KUKA KRL program: MyProgram_318().src

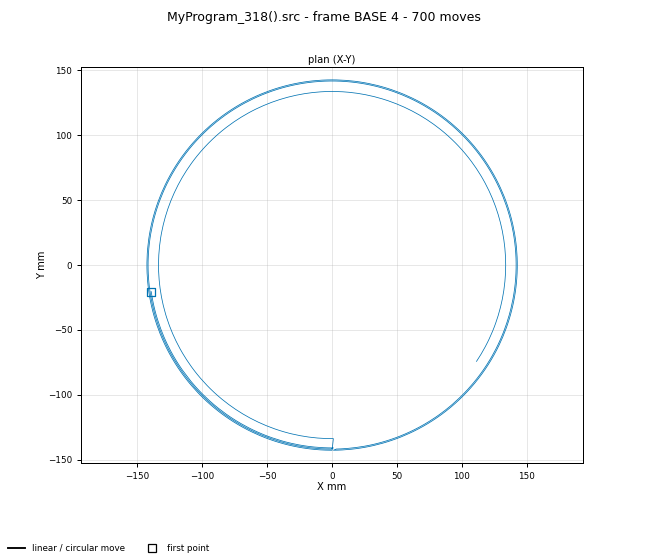
[picture p0: tool path of MyProgram_318().src in frame BASE 4, 700 of 700 moves have a stored position in this frame; points joined in program order, loops and branches not executed]
&ACCESS RVP
&REL 1
&PARAM TEMPLATE = C:\KRC\Roboter\Template\vorgabe
&PARAM EDITMASK = *
DEF MyProgram_318()
; ---- Setting reference (Base) ----
$BASE = BASE_DATA[4]

; --------------------------
; ---- Setting tool (TCP) ----
$TOOL = TOOL_DATA[3]
; --------------------------

$VEL.CP = VEL_APROX_PRINT
Startdeposition()
$VEL.CP = VEL_PRINT
LIN {X -139.4238,Y -20.4254,Z 184,A -166.8954,B 3.5696,C 0.2176,E1 3.4184,E2 259.9212} C_DIS
LIN {X -138.3795,Y -26.5906,Z 184,A -165.0587,B 3.569,C 0.2283,E1 3.4193,E2 258.1802} C_DIS
LIN {X -137.4826,Y -30.8981,Z 184,A -163.1795,B 3.5687,C 0.2327,E1 3.4204,E2 256.2901} C_DIS
LIN {X -136.525,Y -34.8838,Z 184,A -161.5232,B 3.5684,C 0.2373,E1 3.4215,E2 254.636} C_DIS
LIN {X -135.6376,Y -38.1888,Z 184,A -160.0373,B 3.5682,C 0.2406,E1 3.4226,E2 253.1383} C_DIS
LIN {X -134.4577,Y -42.1612,Z 184,A -158.3509,B 3.5678,C 0.2451,E1 3.424,E2 251.4527} C_DIS
LIN {X -131.9427,Y -49.4671,Z 184,A -155.0815,B 3.5673,C 0.2527,E1 3.4271,E2 248.1679} C_DIS
LIN {X -130.7547,Y -52.527,Z 184,A -153.7556,B 3.5671,C 0.2562,E1 3.4284,E2 246.8439} C_DIS
LIN {X -129.4822,Y -55.5908,Z 184,A -152.0943,B 3.5669,C 0.258,E1 3.4303,E2 245.1414} C_DIS
LIN {X -127.3573,Y -60.3009,Z 184,A -150.0342,B 3.5665,C 0.2635,E1 3.4327,E2 243.0877} C_DIS
LIN {X -125.7132,Y -63.6562,Z 184,A -148.6523,B 3.5662,C 0.2681,E1 3.4344,E2 241.7248} C_DIS
LIN {X -124.3831,Y -66.2218,Z 184,A -146.8432,B 3.5662,C 0.2674,E1 3.4368,E2 239.831} C_DIS
LIN {X -122.4083,Y -69.8041,Z 184,A -145.4884,B 3.5658,C 0.2732,E1 3.4386,E2 238.5184} C_DIS
LIN {X -120.1357,Y -73.6466,Z 184,A -143.7295,B 3.5655,C 0.2778,E1 3.4412,E2 236.7677} C_DIS
LIN {X -117.9556,Y -77.0913,Z 184,A -141.8449,B 3.5653,C 0.2803,E1 3.444,E2 234.8531} C_DIS
LIN {X -115.3684,Y -80.9115,Z 184,A -139.9945,B 3.5649,C 0.2847,E1 3.447,E2 233.0067} C_DIS
LIN {X -108.8404,Y -89.5006,Z 184,A -135.5865,B 3.5641,C 0.2942,E1 3.4545,E2 228.5975} C_DIS
LIN {X -105.2184,Y -93.7317,Z 184,A -133.038,B 3.5639,C 0.2971,E1 3.4592,E2 226.0111} C_DIS
LIN {X -102.625,Y -96.5637,Z 184,A -131.4587,B 3.5637,C 0.3001,E1 3.4622,E2 224.4297} C_DIS
LIN {X -99.7736,Y -99.5073,Z 184,A -128.8184,B 3.5639,C 0.2971,E1 3.4678,E2 221.6564} C_DIS
LIN {X -94.4634,Y -104.5617,Z 184,A -126.9429,B 3.5628,C 0.3096,E1 3.4713,E2 219.9326} C_DIS
LIN {X -90.9298,Y -107.6493,Z 184,A -124.7172,B 3.5628,C 0.3109,E1 3.4761,E2 217.664} C_DIS
LIN {X -87.4156,Y -110.5219,Z 184,A -122.849,B 3.5625,C 0.3138,E1 3.4801,E2 215.7928} C_DIS
LIN {X -81.7858,Y -114.7499,Z 184,A -119.9297,B 3.5621,C 0.3179,E1 3.4867,E2 212.866} C_DIS
LIN {X -78.0793,Y -117.3033,Z 184,A -118.0516,B 3.5619,C 0.3203,E1 3.4911,E2 210.9813} C_DIS
LIN {X -74.1308,Y -119.8381,Z 184,A -116.0901,B 3.5617,C 0.3226,E1 3.4957,E2 209.0125} C_DIS
LIN {X -70.4469,Y -122.0396,Z 184,A -114.3288,B 3.5615,C 0.3247,E1 3.5,E2 207.2488} C_DIS
LIN {X -64.5086,Y -125.2793,Z 184,A -111.5655,B 3.5612,C 0.328,E1 3.5068,E2 204.4835} C_DIS
LIN {X -61.1095,Y -126.971,Z 184,A -110.0392,B 3.561,C 0.3298,E1 3.5106,E2 202.9594} C_DIS
LIN {X -57.8227,Y -128.5009,Z 184,A -108.3988,B 3.561,C 0.3301,E1 3.5149,E2 201.296} C_DIS
LIN {X -53.0992,Y -130.5241,Z 184,A -106.388,B 3.5608,C 0.3327,E1 3.52,E2 199.2957} C_DIS
LIN {X -49.9078,Y -131.7776,Z 184,A -105.1272,B 3.5606,C 0.3349,E1 3.5232,E2 198.0529} C_DIS
LIN {X -46.236,Y -133.1094,Z 184,A -102.9524,B 3.5609,C 0.3317,E1 3.5292,E2 195.797} C_DIS
LIN {X -42.002,Y -134.5078,Z 184,A -101.4553,B 3.5605,C 0.3354,E1 3.5331,E2 194.3432} C_DIS
LIN {X -39.0569,Y -135.3911,Z 184,A -100.1869,B 3.5605,C 0.3361,E1 3.5365,E2 193.0719} C_DIS
LIN {X -35.4176,Y -136.3895,Z 184,A -98.6921,B 3.5603,C 0.3373,E1 3.5405,E2 191.5822} C_DIS
LIN {X -31.5759,Y -137.3278,Z 184,A -97.2077,B 3.5602,C 0.3391,E1 3.5445,E2 190.1142} C_DIS
LIN {X -28.2117,Y -138.0581,Z 184,A -95.8313,B 3.5601,C 0.3399,E1 3.5483,E2 188.7406} C_DIS
LIN {X -25.433,Y -138.5982,Z 184,A -94.5046,B 3.5601,C 0.3389,E1 3.552,E2 187.3894} C_DIS
LIN {X -21.5406,Y -139.2549,Z 184,A -92.984,B 3.5601,C 0.34,E1 3.5561,E2 185.8798} C_DIS
LIN {X -17.9488,Y -139.7638,Z 184,A -91.4422,B 3.5601,C 0.3398,E1 3.5604,E2 184.3282} C_DIS
LIN {X -13.5381,Y -140.2594,Z 184,A -89.7378,B 3.56,C 0.3409,E1 3.5651,E2 182.637} C_DIS
LIN {X -10.3708,Y -140.5291,Z 184,A -88.4486,B 3.56,C 0.341,E1 3.5687,E2 181.3477} C_DIS
LIN {X -7.0582,Y -140.7344,Z 184,A -86.9885,B 3.56,C 0.3401,E1 3.5728,E2 179.8718} C_DIS
LIN {X -2.6126,Y -140.8874,Z 184,A -85.2158,B 3.56,C 0.3403,E1 3.5778,E2 178.1032} C_DIS
LIN {X 0.9985,Y -140.9073,Z 184,A -84.3874,B 3.5595,C 0.3456,E1 3.5799,E2 177.3618} C_DIS
Enddeposition()
LIN {X 0.9985,Y -140.9073,Z 184,A -84.3874,B 3.5595,C 0.3456,E1 3.5799,E2 177.3618} C_DIS
Startdeposition()
$VEL.CP = VEL_PRINT
LIN {X -0.7581,Y -141.8102,Z 184,A -85.1116,B 3.5589,C 0.3478,E1 3.5773,E2 178.1199} C_DIS
LIN {X -5.0897,Y -141.7215,Z 184,A -86.9297,B 3.5589,C 0.3485,E1 3.5722,E2 179.9481} C_DIS
LIN {X -9.2783,Y -141.5094,Z 184,A -88.6221,B 3.5589,C 0.3485,E1 3.5675,E2 181.641} C_DIS
LIN {X -13.6823,Y -141.1505,Z 184,A -90.3059,B 3.5589,C 0.3474,E1 3.5628,E2 183.3115} C_DIS
LIN {X -17.2016,Y -140.7655,Z 184,A -91.7391,B 3.5589,C 0.3472,E1 3.5588,E2 184.7456} C_DIS
LIN {X -20.6522,Y -140.3014,Z 184,A -93.2844,B 3.5589,C 0.348,E1 3.5545,E2 186.3106} C_DIS
LIN {X -24.9177,Y -139.6056,Z 184,A -94.9566,B 3.5589,C 0.3468,E1 3.5499,E2 187.9732} C_DIS
LIN {X -28.2573,Y -138.9681,Z 184,A -96.3278,B 3.559,C 0.3463,E1 3.5462,E2 189.3445} C_DIS
LIN {X -32.2456,Y -138.0988,Z 184,A -97.9298,B 3.5591,C 0.3451,E1 3.5418,E2 190.9406} C_DIS
LIN {X -35.6192,Y -137.2678,Z 184,A -99.4409,B 3.5591,C 0.3451,E1 3.5377,E2 192.4668} C_DIS
LIN {X -40.243,Y -135.9825,Z 184,A -101.1414,B 3.5594,C 0.3421,E1 3.5332,E2 194.1351} C_DIS
LIN {X -46.7478,Y -133.8854,Z 184,A -104.5205,B 3.5592,C 0.3448,E1 3.524,E2 197.5994} C_DIS
LIN {X -50.6351,Y -132.4661,Z 184,A -105.7791,B 3.5596,C 0.3403,E1 3.5209,E2 198.802} C_DIS
LIN {X -53.5532,Y -131.3123,Z 184,A -107.0843,B 3.5596,C 0.3394,E1 3.5175,E2 200.1125} C_DIS
LIN {X -56.8322,Y -129.9269,Z 184,A -108.5455,B 3.5598,C 0.3381,E1 3.5137,E2 201.5771} C_DIS
LIN {X -59.8555,Y -128.5612,Z 184,A -109.9347,B 3.5599,C 0.3371,E1 3.5102,E2 202.9731} C_DIS
LIN {X -63.1305,Y -126.9853,Z 184,A -111.4004,B 3.5601,C 0.3354,E1 3.5065,E2 204.4386} C_DIS
LIN {X -66.721,Y -125.1383,Z 184,A -113.2184,B 3.5601,C 0.3349,E1 3.5019,E2 206.2823} C_DIS
LIN {X -70.8009,Y -122.8756,Z 184,A -115.1047,B 3.5603,C 0.3325,E1 3.4973,E2 208.1689} C_DIS
LIN {X -74.881,Y -120.4323,Z 184,A -117.0229,B 3.5606,C 0.3299,E1 3.4927,E2 210.0867} C_DIS
LIN {X -78.6833,Y -117.9832,Z 184,A -118.8829,B 3.5608,C 0.3275,E1 3.4884,E2 211.9511} C_DIS
LIN {X -82.4224,Y -115.4021,Z 184,A -120.7734,B 3.561,C 0.3251,E1 3.484,E2 213.8491} C_DIS
LIN {X -86.4102,Y -112.4477,Z 184,A -122.695,B 3.5614,C 0.3213,E1 3.4798,E2 215.7593} C_DIS
LIN {X -89.4085,Y -110.079,Z 184,A -124.4431,B 3.5614,C 0.3201,E1 3.4759,E2 217.5349} C_DIS
LIN {X -93.1808,Y -106.9039,Z 184,A -126.2519,B 3.5619,C 0.3155,E1 3.4721,E2 219.3188} C_DIS
LIN {X -95.7019,Y -104.6536,Z 184,A -127.8582,B 3.5619,C 0.3145,E1 3.4687,E2 220.9575} C_DIS
LIN {X -100.0347,Y -100.5194,Z 184,A -129.9787,B 3.5625,C 0.3082,E1 3.4645,E2 223.0372} C_DIS
LIN {X -103.5928,Y -96.8488,Z 184,A -132.3732,B 3.5627,C 0.3062,E1 3.4598,E2 225.4759} C_DIS
LIN {X -106.2873,Y -93.8834,Z 184,A -134.2151,B 3.5629,C 0.3042,E1 3.4563,E2 227.3476} C_DIS
LIN {X -109.471,Y -90.1518,Z 184,A -136.1691,B 3.5632,C 0.2999,E1 3.4528,E2 229.2974} C_DIS
LIN {X -112.3501,Y -86.5374,Z 184,A -138.4908,B 3.5633,C 0.2986,E1 3.4487,E2 231.6796} C_DIS
LIN {X -114.9652,Y -83.0311,Z 184,A -139.6861,B 3.5639,C 0.2913,E1 3.4469,E2 232.7977} C_DIS
LIN {X -116.9685,Y -80.184,Z 184,A -141.3736,B 3.5641,C 0.2898,E1 3.4441,E2 234.5225} C_DIS
LIN {X -119.5805,Y -76.2344,Z 184,A -143.3398,B 3.5644,C 0.2857,E1 3.4411,E2 236.4953} C_DIS
LIN {X -121.8868,Y -72.4895,Z 184,A -145.1675,B 3.5647,C 0.2818,E1 3.4385,E2 238.3292} C_DIS
LIN {X -124.1077,Y -68.6177,Z 184,A -147.1404,B 3.565,C 0.2784,E1 3.4357,E2 240.324} C_DIS
LIN {X -125.7385,Y -65.5782,Z 184,A -148.4282,B 3.5653,C 0.2744,E1 3.4341,E2 241.5971} C_DIS
LIN {X -127.3592,Y -62.3725,Z 184,A -149.9746,B 3.5655,C 0.2713,E1 3.4321,E2 243.1556} C_DIS
LIN {X -129.5232,Y -57.7435,Z 184,A -152.0254,B 3.5659,C 0.266,E1 3.4298,E2 245.2037} C_DIS
LIN {X -131.0036,Y -54.3023,Z 184,A -153.6597,B 3.5662,C 0.2628,E1 3.428,E2 246.8533} C_DIS
LIN {X -132.4612,Y -50.6478,Z 184,A -155.2899,B 3.5664,C 0.2588,E1 3.4263,E2 248.4883} C_DIS
LIN {X -133.7803,Y -47.0508,Z 184,A -157.1342,B 3.5666,C 0.2563,E1 3.4245,E2 250.3712} C_DIS
LIN {X -135.5727,Y -41.6009,Z 184,A -159.3512,B 3.5671,C 0.2496,E1 3.4227,E2 252.5735} C_DIS
LIN {X -136.6568,Y -37.8891,Z 184,A -160.9424,B 3.5674,C 0.2456,E1 3.4214,E2 254.1677} C_DIS
LIN {X -137.5543,Y -34.4901,Z 184,A -162.3548,B 3.5677,C 0.2417,E1 3.4204,E2 255.5783} C_DIS
LIN {X -138.2758,Y -31.4708,Z 184,A -163.6845,B 3.5679,C 0.2386,E1 3.4196,E2 256.9172} C_DIS
LIN {X -138.9436,Y -28.3779,Z 184,A -165.4551,B 3.5679,C 0.2376,E1 3.4186,E2 258.752} C_DIS
LIN {X -139.7115,Y -24.3262,Z 184,A -166.9229,B 3.5683,C 0.232,E1 3.4179,E2 260.1928} C_DIS
LIN {X -140.4101,Y -19.891,Z 184,A -168.6787,B 3.5686,C 0.2267,E1 3.4171,E2 261.9398} C_DIS
LIN {X -140.9297,Y -15.8077,Z 184,A -170.7984,B 3.5688,C 0.2243,E1 3.4164,E2 264.1183} C_DIS
LIN {X -141.3049,Y -11.9832,Z 184,A -172.0737,B 3.5691,C 0.2186,E1 3.4161,E2 265.3564} C_DIS
LIN {X -141.646,Y -6.8675,Z 184,A -174.0827,B 3.5695,C 0.2124,E1 3.4158,E2 267.3558} C_DIS
LIN {X -141.7651,Y -3.6623,Z 184,A -175.5929,B 3.5697,C 0.2098,E1 3.4157,E2 268.8933} C_DIS
LIN {X -141.8131,Y 0.1767,Z 184,A -177.0204,B 3.57,C 0.2048,E1 3.4157,E2 270.3036} C_DIS
LIN {X -141.7682,Y 3.5529,Z 184,A -178.6647,B 3.57,C 0.2024,E1 3.4157,E2 271.9835} C_DIS
LIN {X -141.5831,Y 8.0813,Z 184,A 179.6286,B 3.5704,C 0.1966,E1 3.4159,E2 273.6727} C_DIS
LIN {X -141.239,Y 12.7605,Z 184,A 177.393,B 3.5706,C 0.193,E1 3.4165,E2 275.9514} C_DIS
LIN {X -140.7795,Y 17.0836,Z 184,A 175.767,B 3.5709,C 0.1874,E1 3.417,E2 277.559} C_DIS
LIN {X -140.3004,Y 20.659,Z 184,A 174.0083,B 3.571,C 0.1848,E1 3.4177,E2 279.3558} C_DIS
LIN {X -139.7122,Y 24.3224,Z 184,A 172.7327,B 3.5713,C 0.1795,E1 3.4182,E2 280.6013} C_DIS
LIN {X -138.1438,Y 32.0486,Z 184,A 169.8477,B 3.5718,C 0.1692,E1 3.4198,E2 283.4451} C_DIS
LIN {X -137.0717,Y 36.3588,Z 184,A 167.4127,B 3.5718,C 0.1675,E1 3.4215,E2 285.9619} C_DIS
LIN {X -136.0472,Y 40.0221,Z 184,A 165.8748,B 3.5721,C 0.1634,E1 3.4227,E2 287.4988} C_DIS
LIN {X -135.0231,Y 43.3519,Z 184,A 164.3959,B 3.5722,C 0.1599,E1 3.4239,E2 288.9859} C_DIS
LIN {X -133.8089,Y 46.9684,Z 184,A 162.8175,B 3.5724,C 0.156,E1 3.4254,E2 290.5678} C_DIS
LIN {X -132.5738,Y 50.3504,Z 184,A 161.3061,B 3.5726,C 0.1525,E1 3.4269,E2 292.0854} C_DIS
LIN {X -131.2818,Y 53.6289,Z 184,A 159.8333,B 3.5727,C 0.149,E1 3.4284,E2 293.5634} C_DIS
LIN {X -130.0287,Y 56.5967,Z 184,A 158.4531,B 3.5728,C 0.146,E1 3.4299,E2 294.9527} C_DIS
LIN {X -128.4997,Y 59.9885,Z 184,A 156.9056,B 3.573,C 0.1424,E1 3.4317,E2 296.5047} C_DIS
LIN {X -127.0221,Y 63.0558,Z 184,A 155.4507,B 3.5731,C 0.1393,E1 3.4335,E2 297.9686} C_DIS
LIN {X -124.9043,Y 67.1567,Z 184,A 153.6487,B 3.5733,C 0.1344,E1 3.4358,E2 299.7612} C_DIS
LIN {X -123.1361,Y 70.3464,Z 184,A 151.9399,B 3.5733,C 0.132,E1 3.4382,E2 301.4989} C_DIS
LIN {X -120.8558,Y 74.1956,Z 184,A 150.0674,B 3.5735,C 0.128,E1 3.4409,E2 303.3783} C_DIS
LIN {X -118.5023,Y 77.8994,Z 184,A 148.0646,B 3.5736,C 0.1251,E1 3.444,E2 305.4089} C_DIS
LIN {X -115.6188,Y 82.1194,Z 184,A 146.0636,B 3.5738,C 0.12,E1 3.4472,E2 307.4001} C_DIS
LIN {X -112.9327,Y 85.7759,Z 184,A 144.1658,B 3.5739,C 0.1163,E1 3.4504,E2 309.3047} C_DIS
LIN {X -110.048,Y 89.4466,Z 184,A 142.3457,B 3.5741,C 0.1118,E1 3.4535,E2 311.1149} C_DIS
LIN {X -107.6501,Y 92.3182,Z 184,A 140.6682,B 3.5741,C 0.1095,E1 3.4566,E2 312.8123} C_DIS
LIN {X -104.3096,Y 96.0761,Z 184,A 138.8317,B 3.5743,C 0.1043,E1 3.46,E2 314.6225} C_DIS
LIN {X -102.1234,Y 98.3973,Z 184,A 137.2326,B 3.5743,C 0.1034,E1 3.4631,E2 316.26} C_DIS
LIN {X -98.7745,Y 101.7581,Z 184,A 135.333,B 3.5744,C 0.0996,E1 3.4669,E2 318.1559} C_DIS
LIN {X -95.6925,Y 104.6622,Z 184,A 133.5206,B 3.5745,C 0.097,E1 3.4706,E2 319.9798} C_DIS
LIN {X -93.0387,Y 107.0279,Z 184,A 132.0732,B 3.5745,C 0.0945,E1 3.4737,E2 321.4276} C_DIS
LIN {X -89.5567,Y 109.9579,Z 184,A 130.1655,B 3.5746,C 0.0917,E1 3.4778,E2 323.3426} C_DIS
LIN {X -85.9082,Y 112.8316,Z 184,A 128.3025,B 3.5747,C 0.0885,E1 3.4819,E2 325.2025} C_DIS
LIN {X -82.2961,Y 115.4924,Z 184,A 126.3982,B 3.5747,C 0.0861,E1 3.4862,E2 327.1171} C_DIS
LIN {X -78.4994,Y 118.106,Z 184,A 124.612,B 3.5749,C 0.0828,E1 3.4903,E2 328.8923} C_DIS
LIN {X -75.2879,Y 120.1791,Z 184,A 122.8858,B 3.5749,C 0.0817,E1 3.4945,E2 330.6403} C_DIS
LIN {X -70.6565,Y 122.9592,Z 184,A 120.7996,B 3.5749,C 0.0781,E1 3.4994,E2 332.7129} C_DIS
LIN {X -67.3455,Y 124.8028,Z 184,A 119.1375,B 3.5749,C 0.077,E1 3.5036,E2 334.3904} C_DIS
LIN {X -63.8671,Y 126.6167,Z 184,A 117.3142,B 3.5749,C 0.0766,E1 3.5082,E2 336.2424} C_DIS
LIN {X -60.8905,Y 128.074,Z 184,A 116.2429,B 3.5751,C 0.0734,E1 3.5108,E2 337.2792} C_DIS
LIN {X -57.6601,Y 129.5605,Z 184,A 114.759,B 3.5751,C 0.0721,E1 3.5146,E2 338.7681} C_DIS
LIN {X -54.3227,Y 130.9951,Z 184,A 113.2583,B 3.5751,C 0.0708,E1 3.5184,E2 340.272} C_DIS
LIN {X -50.7357,Y 132.427,Z 184,A 111.1717,B 3.5751,C 0.073,E1 3.5241,E2 342.4234} C_DIS
LIN {X -46.357,Y 134.0209,Z 184,A 109.7766,B 3.5751,C 0.068,E1 3.5276,E2 343.7564} C_DIS
LIN {X -42.4916,Y 135.2979,Z 184,A 108.1605,B 3.5751,C 0.0665,E1 3.5319,E2 345.368} C_DIS
LIN {X -39.0206,Y 136.3403,Z 184,A 106.3392,B 3.5751,C 0.068,E1 3.5369,E2 347.2332} C_DIS
LIN {X -35.6094,Y 137.2702,Z 184,A 105.2757,B 3.5752,C 0.0645,E1 3.5396,E2 348.2501} C_DIS
LIN {X -31.0466,Y 138.3727,Z 184,A 103.3247,B 3.5752,C 0.0639,E1 3.5449,E2 350.2069} C_DIS
LIN {X -27.2162,Y 139.1771,Z 184,A 101.1819,B 3.5752,C 0.0673,E1 3.551,E2 352.419} C_DIS
LIN {X -22.493,Y 140.0187,Z 184,A 99.5827,B 3.5752,C 0.064,E1 3.5553,E2 353.9748} C_DIS
LIN {X -17.751,Y 140.6983,Z 184,A 97.7622,B 3.5752,C 0.0626,E1 3.5603,E2 355.78} C_DIS
LIN {X -13.7012,Y 141.1487,Z 184,A 96.1311,B 3.5752,C 0.0622,E1 3.5648,E2 357.4083} C_DIS
LIN {X -9.471,Y 141.4975,Z 184,A 94.2713,B 3.5752,C 0.0631,E1 3.57,E2 359.2855} C_DIS
LIN {X -5.7272,Y 141.6966,Z 184,A 92.8784,B 3.5752,C 0.0621,E1 3.5739,E2 360.6624} C_DIS
LIN {X -1.3489,Y 141.8069,Z 184,A 91.1035,B 3.5752,C 0.0623,E1 3.5789,E2 362.4373} C_DIS
LIN {X 2.3537,Y 141.7926,Z 184,A 89.6494,B 3.5752,C 0.0621,E1 3.5829,E2 363.8855} C_DIS
LIN {X 6.5238,Y 141.6632,Z 184,A 87.8816,B 3.5752,C 0.0631,E1 3.5879,E2 365.6629} C_DIS
LIN {X 10.4865,Y 141.4239,Z 184,A 86.3928,B 3.5752,C 0.0626,E1 3.592,E2 367.1366} C_DIS
LIN {X 14.6588,Y 141.0533,Z 184,A 84.6233,B 3.5752,C 0.0639,E1 3.5969,E2 368.9152} C_DIS
LIN {X 18.435,Y 140.6086,Z 184,A 83.1856,B 3.5752,C 0.0638,E1 3.6009,E2 370.34} C_DIS
LIN {X 22.252,Y 140.0564,Z 184,A 81.6384,B 3.5752,C 0.0645,E1 3.6051,E2 371.8853} C_DIS
LIN {X 25.9323,Y 139.4225,Z 184,A 80.0467,B 3.5752,C 0.0661,E1 3.6096,E2 373.487} C_DIS
LIN {X 30.0417,Y 138.5933,Z 184,A 78.4442,B 3.5752,C 0.0664,E1 3.6139,E2 375.0775} C_DIS
LIN {X 34.067,Y 137.6616,Z 184,A 76.5458,B 3.5752,C 0.0697,E1 3.6191,E2 377.0043} C_DIS
LIN {X 37.236,Y 136.8378,Z 184,A 75.5319,B 3.5752,C 0.0681,E1 3.6218,E2 377.9791} C_DIS
LIN {X 43.0876,Y 135.1075,Z 184,A 72.6176,B 3.575,C 0.0743,E1 3.6297,E2 380.9492} C_DIS
LIN {X 47.3667,Y 133.6696,Z 184,A 71.319,B 3.5751,C 0.0714,E1 3.633,E2 382.1814} C_DIS
LIN {X 50.32,Y 132.5852,Z 184,A 70.0377,B 3.5751,C 0.0729,E1 3.6363,E2 383.4638} C_DIS
LIN {X 53.5602,Y 131.3095,Z 184,A 68.6098,B 3.5751,C 0.0747,E1 3.64,E2 384.8941} C_DIS
LIN {X 56.7669,Y 129.9551,Z 184,A 67.2856,B 3.5751,C 0.0756,E1 3.6434,E2 386.2078} C_DIS
LIN {X 59.8342,Y 128.5711,Z 184,A 65.8968,B 3.575,C 0.0776,E1 3.6469,E2 387.6001} C_DIS
LIN {X 63.2915,Y 126.9058,Z 184,A 64.4015,B 3.575,C 0.0791,E1 3.6507,E2 389.0883} C_DIS
LIN {X 66.8063,Y 125.0925,Z 184,A 62.7191,B 3.5749,C 0.0821,E1 3.6549,E2 390.7813} C_DIS
LIN {X 70.8243,Y 122.8621,Z 184,A 60.9061,B 3.5749,C 0.0844,E1 3.6593,E2 392.5886} C_DIS
LIN {X 74.6858,Y 120.5538,Z 184,A 59.1267,B 3.5748,C 0.0868,E1 3.6635,E2 394.3632} C_DIS
LIN {X 78.4315,Y 118.1513,Z 184,A 57.4145,B 3.5748,C 0.0889,E1 3.6675,E2 396.0646} C_DIS
LIN {X 81.9336,Y 115.7499,Z 184,A 55.6871,B 3.5746,C 0.0919,E1 3.6714,E2 397.7934} C_DIS
LIN {X 84.8953,Y 113.5955,Z 184,A 54.2829,B 3.5746,C 0.0937,E1 3.6746,E2 399.1881} C_DIS
LIN {X 88.4894,Y 110.8187,Z 184,A 52.4477,B 3.5746,C 0.097,E1 3.6786,E2 401.0235} C_DIS
LIN {X 92.1059,Y 107.8318,Z 184,A 50.6397,B 3.5744,C 0.0997,E1 3.6824,E2 402.8206} C_DIS
LIN {X 95.439,Y 104.8929,Z 184,A 48.8214,B 3.5744,C 0.1034,E1 3.6862,E2 404.642} C_DIS
LIN {X 98.8945,Y 101.642,Z 184,A 47.024,B 3.5742,C 0.106,E1 3.6898,E2 406.4245} C_DIS
LIN {X 102.1017,Y 98.4196,Z 184,A 45.2316,B 3.5742,C 0.1093,E1 3.6933,E2 408.2115} C_DIS
LIN {X 105.1426,Y 95.1639,Z 184,A 43.493,B 3.574,C 0.1125,E1 3.6966,E2 409.9426} C_DIS
LIN {X 108.1815,Y 91.6946,Z 184,A 41.6738,B 3.574,C 0.1161,E1 3.6999,E2 411.7566} C_DIS
LIN {X 111.1562,Y 88.0653,Z 184,A 39.7825,B 3.5738,C 0.1203,E1 3.7032,E2 413.6478} C_DIS
LIN {X 113.9616,Y 84.4037,Z 184,A 38.0457,B 3.5737,C 0.1232,E1 3.7061,E2 415.3687} C_DIS
LIN {X 116.6457,Y 80.6539,Z 184,A 36.2393,B 3.5736,C 0.127,E1 3.709,E2 417.1684} C_DIS
LIN {X 119.0779,Y 77.017,Z 184,A 34.5492,B 3.5734,C 0.1303,E1 3.7116,E2 418.8491} C_DIS
LIN {X 121.3791,Y 73.3363,Z 184,A 32.8628,B 3.5734,C 0.1339,E1 3.7141,E2 420.5273} C_DIS
LIN {X 123.5885,Y 69.5484,Z 184,A 31.1169,B 3.5732,C 0.138,E1 3.7165,E2 422.2705} C_DIS
LIN {X 125.7362,Y 65.5825,Z 184,A 29.454,B 3.573,C 0.1408,E1 3.7186,E2 423.9134} C_DIS
LIN {X 127.3091,Y 62.4741,Z 184,A 28.0813,B 3.573,C 0.144,E1 3.7203,E2 425.2823} C_DIS
LIN {X 128.8911,Y 59.1422,Z 184,A 26.6443,B 3.5728,C 0.1472,E1 3.722,E2 426.713} C_DIS
LIN {X 130.3679,Y 55.8122,Z 184,A 25.2416,B 3.5727,C 0.1503,E1 3.7236,E2 428.1074} C_DIS
LIN {X 131.7718,Y 52.4133,Z 184,A 23.8217,B 3.5725,C 0.1535,E1 3.7251,E2 429.5194} C_DIS
LIN {X 133.0746,Y 49.0132,Z 184,A 22.3927,B 3.5724,C 0.1569,E1 3.7265,E2 430.9436} C_DIS
LIN {X 134.2106,Y 45.8097,Z 184,A 21.0727,B 3.5722,C 0.16,E1 3.7277,E2 432.2573} C_DIS
LIN {X 135.2039,Y 42.7857,Z 184,A 19.7954,B 3.5721,C 0.1634,E1 3.7288,E2 433.5341} C_DIS
LIN {X 136.5763,Y 38.1771,Z 184,A 17.9257,B 3.5719,C 0.1678,E1 3.7302,E2 435.3953} C_DIS
LIN {X 137.5376,Y 34.5558,Z 184,A 16.4903,B 3.5717,C 0.1711,E1 3.7312,E2 436.8213} C_DIS
LIN {X 138.4117,Y 30.8758,Z 184,A 14.9257,B 3.5715,C 0.1757,E1 3.7322,E2 438.3916} C_DIS
LIN {X 139.5625,Y 25.1588,Z 184,A 12.7711,B 3.5713,C 0.18,E1 3.7333,E2 440.521} C_DIS
LIN {X 140.1862,Y 21.4138,Z 184,A 11.2596,B 3.5711,C 0.184,E1 3.734,E2 442.0304} C_DIS
LIN {X 140.7594,Y 17.2527,Z 184,A 9.5729,B 3.5708,C 0.1886,E1 3.7346,E2 443.7168} C_DIS
LIN {X 141.1688,Y 13.4917,Z 184,A 8.1633,B 3.5707,C 0.1916,E1 3.735,E2 445.1117} C_DIS
LIN {X 141.495,Y 9.5104,Z 184,A 6.4959,B 3.5704,C 0.1967,E1 3.7354,E2 446.7873} C_DIS
LIN {X 141.7161,Y 5.2276,Z 184,A 4.9188,B 3.5702,C 0.1999,E1 3.7356,E2 448.345} C_DIS
LIN {X 141.8087,Y 1.0186,Z 184,A 3.3066,B 3.57,C 0.2037,E1 3.7356,E2 449.9465} C_DIS
LIN {X 141.7901,Y -2.5054,Z 184,A 1.951,B 3.5698,C 0.2069,E1 3.7356,E2 451.2942} C_DIS
LIN {X 141.6567,Y -6.6532,Z 184,A 0.2503,B 3.5695,C 0.2119,E1 3.7354,E2 452.9992} C_DIS
LIN {X 141.4207,Y -10.5304,Z 184,A -1.1819,B 3.5694,C 0.2148,E1 3.7351,E2 454.4143} C_DIS
LIN {X 141.0452,Y -14.7346,Z 184,A -2.9015,B 3.5691,C 0.2198,E1 3.7347,E2 456.137} C_DIS
LIN {X 140.6026,Y -18.4812,Z 184,A -4.2754,B 3.5689,C 0.2223,E1 3.7342,E2 457.492} C_DIS
LIN {X 140.0659,Y -22.1904,Z 184,A -5.7496,B 3.5687,C 0.2261,E1 3.7336,E2 458.9621} C_DIS
LIN {X 139.3696,Y -26.2089,Z 184,A -7.3723,B 3.5684,C 0.2304,E1 3.7328,E2 460.5826} C_DIS
LIN {X 138.4697,Y -30.6145,Z 184,A -9.0357,B 3.5682,C 0.2337,E1 3.7318,E2 462.227} C_DIS
LIN {X 137.8173,Y -33.422,Z 184,A -10.1817,B 3.568,C 0.2367,E1 3.7311,E2 463.3714} C_DIS
LIN {X 136.4961,Y -38.464,Z 184,A -12.2228,B 3.5676,C 0.2418,E1 3.7296,E2 465.4054} C_DIS
LIN {X 134.6511,Y -44.4944,Z 184,A -14.8786,B 3.5671,C 0.2499,E1 3.7274,E2 468.0777} C_DIS
LIN {X 132.5838,Y -50.3236,Z 184,A -17.0608,B 3.5669,C 0.253,E1 3.7253,E2 470.2195} C_DIS
LIN {X 131.3722,Y -53.4046,Z 184,A -18.3931,B 3.5666,C 0.2565,E1 3.724,E2 471.5522} C_DIS
LIN {X 129.6366,Y -57.49,Z 184,A -20.292,B 3.5662,C 0.2624,E1 3.7218,E2 473.4666} C_DIS
LIN {X 127.7631,Y -61.5412,Z 184,A -21.8421,B 3.5661,C 0.2642,E1 3.72,E2 474.9842} C_DIS
LIN {X 126.2478,Y -64.5917,Z 184,A -23.1637,B 3.5658,C 0.2671,E1 3.7184,E2 476.2996} C_DIS
LIN {X 123.295,Y -70.0678,Z 184,A -25.5094,B 3.5655,C 0.2716,E1 3.7153,E2 478.6248} C_DIS
LIN {X 121.5366,Y -73.076,Z 184,A -27.0493,B 3.5651,C 0.2765,E1 3.713,E2 480.1837} C_DIS
LIN {X 119.1386,Y -76.9235,Z 184,A -28.8197,B 3.5648,C 0.2803,E1 3.7104,E2 481.9473} C_DIS
LIN {X 116.6918,Y -80.5871,Z 184,A -30.5138,B 3.5646,C 0.2836,E1 3.7078,E2 483.6313} C_DIS
LIN {X 114.2062,Y -84.0718,Z 184,A -32.2569,B 3.5642,C 0.2878,E1 3.7049,E2 485.3777} C_DIS
LIN {X 111.9161,Y -87.0974,Z 184,A -33.6922,B 3.564,C 0.2903,E1 3.7025,E2 486.801} C_DIS
LIN {X 109.05,Y -90.6602,Z 184,A -36.2224,B 3.5631,C 0.3018,E1 3.6978,E2 489.4247} C_DIS
LIN {X 104.7171,Y -95.6327,Z 184,A -37.9514,B 3.5634,C 0.2975,E1 3.6948,E2 491.0298} C_DIS
LIN {X 102.145,Y -98.3749,Z 184,A -39.5733,B 3.5631,C 0.3018,E1 3.6916,E2 492.6669} C_DIS
LIN {X 98.3692,Y -102.1506,Z 184,A -41.8051,B 3.5626,C 0.3071,E1 3.6872,E2 494.9105} C_DIS
LIN {X 93.0128,Y -107.0505,Z 184,A -44.2498,B 3.5626,C 0.3077,E1 3.6822,E2 497.2911} C_DIS
LIN {X 90.6834,Y -109.0308,Z 184,A -45.7128,B 3.5622,C 0.3125,E1 3.679,E2 498.7862} C_DIS
LIN {X 87.0751,Y -111.9334,Z 184,A -47.5792,B 3.5619,C 0.3159,E1 3.6749,E2 500.6534} C_DIS
LIN {X 82.6246,Y -115.2575,Z 184,A -49.6349,B 3.5617,C 0.3179,E1 3.6704,E2 502.6851} C_DIS
LIN {X 79.8515,Y -117.1965,Z 184,A -51.6427,B 3.5609,C 0.3268,E1 3.6655,E2 504.7812} C_DIS
LIN {X 75.0709,Y -120.3141,Z 184,A -53.6443,B 3.5609,C 0.3274,E1 3.6609,E2 506.7433} C_DIS
LIN {X 71.3861,Y -122.5368,Z 184,A -55.0283,B 3.5609,C 0.3265,E1 3.6577,E2 508.0803} C_DIS
LIN {X 67.317,Y -124.8181,Z 184,A -56.8303,B 3.5607,C 0.3284,E1 3.6533,E2 509.8725} C_DIS
LIN {X 63.4428,Y -126.8312,Z 184,A -58.4524,B 3.5607,C 0.3295,E1 3.6493,E2 511.4764} C_DIS
LIN {X 60.3215,Y -128.3455,Z 184,A -60.3103,B 3.56,C 0.3359,E1 3.6444,E2 513.3977} C_DIS
LIN {X 56.5063,Y -130.0678,Z 184,A -61.3013,B 3.5605,C 0.3311,E1 3.6421,E2 514.294} C_DIS
LIN {X 52.6238,Y -131.687,Z 184,A -63.2158,B 3.5601,C 0.3353,E1 3.6371,E2 516.2393} C_DIS
LIN {X 49.3829,Y -132.9362,Z 184,A -64.603,B 3.5599,C 0.3367,E1 3.6335,E2 517.6252} C_DIS
LIN {X 44.5518,Y -134.632,Z 184,A -66.6349,B 3.5598,C 0.3386,E1 3.6281,E2 519.6534} C_DIS
LIN {X 40.4313,Y -135.9274,Z 184,A -68.515,B 3.5595,C 0.3415,E1 3.623,E2 521.5533} C_DIS
LIN {X 35.9286,Y -137.1865,Z 184,A -70.1982,B 3.5595,C 0.3412,E1 3.6186,E2 523.2094} C_DIS
LIN {X 32.2158,Y -138.1056,Z 184,A -71.7743,B 3.5594,C 0.3428,E1 3.6143,E2 524.7907} C_DIS
LIN {X 28.5507,Y -138.9084,Z 184,A -73.2669,B 3.5593,C 0.3437,E1 3.6102,E2 526.281} C_DIS
LIN {X 24.7544,Y -139.6348,Z 184,A -74.7465,B 3.5593,C 0.3439,E1 3.6062,E2 527.7502} C_DIS
LIN {X 21.3345,Y -140.1984,Z 184,A -76.4359,B 3.5589,C 0.3474,E1 3.6014,E2 529.4801} C_DIS
LIN {X 18.0595,Y -140.6579,Z 184,A -77.3477,B 3.5592,C 0.3442,E1 3.599,E2 530.3344} C_DIS
LIN {X 14.9692,Y -141.0199,Z 184,A -78.718,B 3.5591,C 0.3459,E1 3.5952,E2 531.721} C_DIS
LIN {X 11.378,Y -141.356,Z 184,A -80.2733,B 3.5589,C 0.3473,E1 3.5908,E2 533.2905} C_DIS
LIN {X 6.9449,Y -141.6421,Z 184,A -81.9498,B 3.5589,C 0.3468,E1 3.5862,E2 534.9517} C_DIS
LIN {X 3.2646,Y -141.7762,Z 184,A -83.5704,B 3.5589,C 0.3483,E1 3.5816,E2 536.5913} C_DIS
LIN {X 3.2646,Y -141.7762,Z 184,A -83.5704,B 3.5589,C 0.3483,E1 3.5816,E2 536.5913} C_DIS
Enddeposition()
LIN {X 1.0052,Y -142.7086,Z 184,A -84.0549,B 3.5589,C 0.3467,E1 3.5802,E2 537.0484} C_DIS
Startdeposition()
$VEL.CP = VEL_PRINT
LIN {X 4.2775,Y -142.6492,Z 184,A -82.4133,B 3.5591,C 0.3435,E1 3.5849,E2 535.3605} C_DIS
LIN {X 7.9235,Y -142.4949,Z 184,A -80.9486,B 3.5591,C 0.3431,E1 3.589,E2 533.8951} C_DIS
LIN {X 11.4177,Y -142.2567,Z 184,A -79.5673,B 3.5592,C 0.3428,E1 3.5928,E2 532.5166} C_DIS
LIN {X 14.817,Y -141.9423,Z 184,A -78.185,B 3.5592,C 0.3421,E1 3.5967,E2 531.1319} C_DIS
LIN {X 18.3077,Y -141.5339,Z 184,A -76.7717,B 3.5594,C 0.3414,E1 3.6006,E2 529.7174} C_DIS
LIN {X 21.7735,Y -141.0421,Z 184,A -75.3977,B 3.5594,C 0.3409,E1 3.6044,E2 528.3471} C_DIS
LIN {X 25.2248,Y -140.4658,Z 184,A -73.9952,B 3.5594,C 0.34,E1 3.6082,E2 526.944} C_DIS
LIN {X 28.7456,Y -139.788,Z 184,A -72.5934,B 3.5595,C 0.3394,E1 3.6121,E2 525.5466} C_DIS
LIN {X 32.1637,Y -139.0416,Z 184,A -71.1939,B 3.5596,C 0.3384,E1 3.6159,E2 524.147} C_DIS
LIN {X 35.5629,Y -138.2114,Z 184,A -69.8118,B 3.5597,C 0.3374,E1 3.6196,E2 522.7671} C_DIS
LIN {X 38.8567,Y -137.3217,Z 184,A -68.451,B 3.5598,C 0.3363,E1 3.6233,E2 521.4067} C_DIS
LIN {X 42.307,Y -136.2987,Z 184,A -67.0228,B 3.56,C 0.335,E1 3.6271,E2 519.9799} C_DIS
LIN {X 45.8165,Y -135.1603,Z 184,A -65.4149,B 3.5602,C 0.3323,E1 3.6314,E2 518.3534} C_DIS
LIN {X 49.7332,Y -133.7669,Z 184,A -63.9217,B 3.5602,C 0.3322,E1 3.6353,E2 516.8835} C_DIS
LIN {X 52.9964,Y -132.5081,Z 184,A -62.541,B 3.5604,C 0.3308,E1 3.6389,E2 515.5051} C_DIS
LIN {X 56.3628,Y -131.1113,Z 184,A -61.0424,B 3.5606,C 0.3286,E1 3.6427,E2 514.0006} C_DIS
LIN {X 59.4446,Y -129.7437,Z 184,A -59.7768,B 3.5606,C 0.3278,E1 3.6459,E2 512.7463} C_DIS
LIN {X 62.5975,Y -128.2527,Z 184,A -58.3023,B 3.5609,C 0.3251,E1 3.6497,E2 511.2605} C_DIS
LIN {X 66.1341,Y -126.4641,Z 184,A -56.8165,B 3.5609,C 0.3239,E1 3.6533,E2 509.7882} C_DIS
LIN {X 69.9862,Y -124.3759,Z 184,A -55.0502,B 3.5612,C 0.3213,E1 3.6577,E2 508.0196} C_DIS
LIN {X 73.7992,Y -122.152,Z 184,A -53.3142,B 3.5614,C 0.3189,E1 3.6618,E2 506.2873} C_DIS
LIN {X 77.4988,Y -119.8392,Z 184,A -51.5917,B 3.5617,C 0.3163,E1 3.6659,E2 504.5675} C_DIS
LIN {X 81.1498,Y -117.3981,Z 184,A -49.8606,B 3.5619,C 0.3137,E1 3.6699,E2 502.8396} C_DIS
LIN {X 84.6977,Y -114.8641,Z 184,A -48.1688,B 3.5621,C 0.3112,E1 3.6737,E2 501.1546} C_DIS
LIN {X 88.1764,Y -112.2156,Z 184,A -46.4638,B 3.5623,C 0.3086,E1 3.6774,E2 499.4551} C_DIS
LIN {X 91.5358,Y -109.4928,Z 184,A -44.7518,B 3.5626,C 0.3055,E1 3.6811,E2 497.7451} C_DIS
LIN {X 94.9015,Y -106.5894,Z 184,A -43.0112,B 3.5629,C 0.3025,E1 3.6848,E2 496.0092} C_DIS
LIN {X 98.1237,Y -103.6302,Z 184,A -41.3219,B 3.5631,C 0.2997,E1 3.6882,E2 494.3277} C_DIS
LIN {X 101.2179,Y -100.6099,Z 184,A -39.6325,B 3.5634,C 0.2967,E1 3.6915,E2 492.6434} C_DIS
LIN {X 104.2456,Y -97.4697,Z 184,A -37.9184,B 3.5636,C 0.2933,E1 3.6948,E2 490.9331} C_DIS
LIN {X 107.1776,Y -94.2365,Z 184,A -36.2155,B 3.5639,C 0.2901,E1 3.698,E2 489.2356} C_DIS
LIN {X 110.0545,Y -90.8596,Z 184,A -34.5118,B 3.5641,C 0.287,E1 3.701,E2 487.5411} C_DIS
LIN {X 112.7909,Y -87.4393,Z 184,A -32.806,B 3.5644,C 0.2835,E1 3.704,E2 485.8411} C_DIS
LIN {X 115.3972,Y -83.9701,Z 184,A -31.1008,B 3.5647,C 0.2799,E1 3.7068,E2 484.1395} C_DIS
LIN {X 117.9157,Y -80.3959,Z 184,A -29.3918,B 3.565,C 0.2762,E1 3.7095,E2 482.4355} C_DIS
LIN {X 120.3272,Y -76.7387,Z 184,A -27.7075,B 3.5653,C 0.2728,E1 3.712,E2 480.76} C_DIS
LIN {X 122.623,Y -73.0139,Z 184,A -26.0232,B 3.5655,C 0.2693,E1 3.7145,E2 479.0842} C_DIS
LIN {X 124.8161,Y -69.1979,Z 184,A -24.3101,B 3.5658,C 0.2655,E1 3.7168,E2 477.377} C_DIS
LIN {X 126.8728,Y -65.3497,Z 184,A -22.581,B 3.5661,C 0.2613,E1 3.719,E2 475.6496} C_DIS
LIN {X 128.6899,Y -61.691,Z 184,A -21.1397,B 3.5663,C 0.2593,E1 3.7208,E2 474.2342} C_DIS
LIN {X 130.1148,Y -58.6272,Z 184,A -19.8114,B 3.5665,C 0.2561,E1 3.7223,E2 472.9087} C_DIS
LIN {X 131.4961,Y -55.4605,Z 184,A -18.4616,B 3.5667,C 0.2529,E1 3.7238,E2 471.5629} C_DIS
LIN {X 132.8489,Y -52.1368,Z 184,A -17.088,B 3.5669,C 0.2499,E1 3.7252,E2 470.1974} C_DIS
LIN {X 134.0672,Y -48.92,Z 184,A -15.7406,B 3.5672,C 0.2466,E1 3.7265,E2 468.8534} C_DIS
LIN {X 135.2256,Y -45.6205,Z 184,A -14.3869,B 3.5674,C 0.2434,E1 3.7277,E2 467.5055} C_DIS
LIN {X 136.4652,Y -41.7629,Z 184,A -12.7702,B 3.5677,C 0.2391,E1 3.7291,E2 465.8888} C_DIS
LIN {X 137.5421,Y -38.0684,Z 184,A -11.3325,B 3.5679,C 0.2361,E1 3.7302,E2 464.4645} C_DIS
LIN {X 138.4382,Y -34.6696,Z 184,A -9.9771,B 3.5681,C 0.2328,E1 3.7311,E2 463.1156} C_DIS
LIN {X 139.2458,Y -31.2696,Z 184,A -8.6275,B 3.5683,C 0.2296,E1 3.732,E2 461.7723} C_DIS
LIN {X 139.9729,Y -27.8372,Z 184,A -7.2751,B 3.5685,C 0.2263,E1 3.7327,E2 460.4264} C_DIS
LIN {X 140.6137,Y -24.3986,Z 184,A -5.9265,B 3.5687,C 0.223,E1 3.7334,E2 459.0843} C_DIS
LIN {X 141.1696,Y -20.9445,Z 184,A -4.5486,B 3.5689,C 0.2194,E1 3.734,E2 457.709} C_DIS
LIN {X 141.6415,Y -17.4628,Z 184,A -3.1978,B 3.5691,C 0.2161,E1 3.7344,E2 456.3653} C_DIS
LIN {X 142.0265,Y -13.984,Z 184,A -1.7891,B 3.5694,C 0.2121,E1 3.7349,E2 454.9551} C_DIS
LIN {X 142.3869,Y -9.6688,Z 184,A -0.1893,B 3.5696,C 0.2088,E1 3.7352,E2 453.3728} C_DIS
LIN {X 142.5807,Y -6.173,Z 184,A 1.3346,B 3.5699,C 0.2035,E1 3.7354,E2 451.8319} C_DIS
LIN {X 142.7037,Y -1.746,Z 184,A 2.9567,B 3.5701,C 0.2003,E1 3.7354,E2 450.2297} C_DIS
LIN {X 142.6935,Y 2.3587,Z 184,A 4.4901,B 3.5702,C 0.197,E1 3.7354,E2 448.7106} C_DIS
LIN {X 142.5808,Y 6.1712,Z 184,A 5.9173,B 3.5704,C 0.1938,E1 3.7353,E2 447.2965} C_DIS
LIN {X 142.387,Y 9.6675,Z 184,A 7.3052,B 3.5706,C 0.1901,E1 3.7351,E2 445.91} C_DIS
LIN {X 142.114,Y 13.0732,Z 184,A 8.6198,B 3.5708,C 0.1869,E1 3.7347,E2 444.6022} C_DIS
LIN {X 141.7492,Y 16.56,Z 184,A 9.9674,B 3.571,C 0.1836,E1 3.7343,E2 443.2618} C_DIS
LIN {X 141.2878,Y 20.1174,Z 184,A 11.3323,B 3.5711,C 0.1804,E1 3.7338,E2 441.9061} C_DIS
LIN {X 140.6097,Y 24.4211,Z 184,A 13.0392,B 3.5713,C 0.176,E1 3.733,E2 440.2038} C_DIS
LIN {X 139.9681,Y 27.8607,Z 184,A 14.3874,B 3.5715,C 0.1728,E1 3.7323,E2 438.8624} C_DIS
LIN {X 139.2435,Y 31.2797,Z 184,A 15.8371,B 3.5717,C 0.1684,E1 3.7315,E2 437.4056} C_DIS
LIN {X 138.2106,Y 35.5664,Z 184,A 17.4274,B 3.5718,C 0.1656,E1 3.7304,E2 435.8384} C_DIS
LIN {X 137.3214,Y 38.8575,Z 184,A 18.783,B 3.572,C 0.162,E1 3.7294,E2 434.4838} C_DIS
LIN {X 136.0493,Y 43.0999,Z 184,A 20.4684,B 3.5722,C 0.1582,E1 3.728,E2 432.8098} C_DIS
LIN {X 134.9512,Y 46.4237,Z 184,A 21.8248,B 3.5723,C 0.155,E1 3.7268,E2 431.4592} C_DIS
LIN {X 133.7678,Y 49.731,Z 184,A 23.1798,B 3.5724,C 0.1519,E1 3.7255,E2 430.1109} C_DIS
LIN {X 132.5086,Y 52.9951,Z 184,A 24.5333,B 3.5726,C 0.1488,E1 3.7241,E2 428.7635} C_DIS
LIN {X 131.1698,Y 56.2274,Z 184,A 25.976,B 3.5727,C 0.1447,E1 3.7226,E2 427.3151} C_DIS
LIN {X 129.7522,Y 59.4262,Z 184,A 27.2409,B 3.5728,C 0.1426,E1 3.7211,E2 426.0682} C_DIS
LIN {X 128.2564,Y 62.5899,Z 184,A 28.6965,B 3.573,C 0.1384,E1 3.7194,E2 424.6053} C_DIS
LIN {X 126.4705,Y 66.122,Z 184,A 30.1605,B 3.573,C 0.1358,E1 3.7175,E2 423.1572} C_DIS
LIN {X 124.3759,Y 69.9861,Z 184,A 31.8976,B 3.5732,C 0.1317,E1 3.7152,E2 421.4231} C_DIS
LIN {X 122.1723,Y 73.7655,Z 184,A 33.6048,B 3.5734,C 0.128,E1 3.7127,E2 419.7218} C_DIS
LIN {X 119.8541,Y 77.4757,Z 184,A 35.3137,B 3.5735,C 0.1242,E1 3.7102,E2 418.0186} C_DIS
LIN {X 117.4231,Y 81.1137,Z 184,A 37.0349,B 3.5736,C 0.1205,E1 3.7075,E2 416.3015} C_DIS
LIN {X 114.877,Y 84.6803,Z 184,A 38.7083,B 3.5737,C 0.1173,E1 3.7048,E2 414.6389} C_DIS
LIN {X 112.2202,Y 88.1705,Z 184,A 40.4084,B 3.5739,C 0.114,E1 3.7019,E2 412.9463} C_DIS
LIN {X 109.4942,Y 91.5342,Z 184,A 42.1149,B 3.5739,C 0.1105,E1 3.6988,E2 411.2436} C_DIS
LIN {X 106.6093,Y 94.8793,Z 184,A 43.8404,B 3.5741,C 0.1072,E1 3.6957,E2 409.524} C_DIS
LIN {X 103.6452,Y 98.1078,Z 184,A 45.5271,B 3.5741,C 0.1042,E1 3.6925,E2 407.8465} C_DIS
LIN {X 100.6014,Y 101.2263,Z 184,A 47.2286,B 3.5742,C 0.1011,E1 3.6891,E2 406.1509} C_DIS
LIN {X 97.4629,Y 104.252,Z 184,A 48.9487,B 3.5743,C 0.098,E1 3.6857,E2 404.4345} C_DIS
LIN {X 94.2233,Y 107.1893,Z 184,A 50.6629,B 3.5744,C 0.095,E1 3.6821,E2 402.7256} C_DIS
LIN {X 90.8612,Y 110.0532,Z 184,A 52.3655,B 3.5744,C 0.0924,E1 3.6785,E2 401.0319} C_DIS
LIN {X 87.4385,Y 112.7915,Z 184,A 54.0963,B 3.5745,C 0.0895,E1 3.6747,E2 399.3048} C_DIS
LIN {X 83.9673,Y 115.3992,Z 184,A 55.8296,B 3.5746,C 0.0866,E1 3.6708,E2 397.5727} C_DIS
LIN {X 80.3917,Y 117.9186,Z 184,A 57.5275,B 3.5746,C 0.0843,E1 3.6669,E2 395.8824} C_DIS
LIN {X 76.7395,Y 120.3267,Z 184,A 59.2284,B 3.5747,C 0.082,E1 3.6629,E2 394.1887} C_DIS
LIN {X 73.016,Y 122.6217,Z 184,A 60.9335,B 3.5747,C 0.0798,E1 3.6589,E2 392.4901} C_DIS
LIN {X 69.009,Y 124.9208,Z 184,A 62.7202,B 3.5748,C 0.0778,E1 3.6545,E2 390.7124} C_DIS
LIN {X 65.3472,Y 126.8741,Z 184,A 64.4312,B 3.5748,C 0.075,E1 3.6503,E2 388.9957} C_DIS
LIN {X 61.8009,Y 128.6374,Z 184,A 65.8779,B 3.5748,C 0.0743,E1 3.6467,E2 387.5676} C_DIS
LIN {X 58.6306,Y 130.1132,Z 184,A 67.2458,B 3.5749,C 0.0729,E1 3.6432,E2 386.2045} C_DIS
LIN {X 55.4638,Y 131.4948,Z 184,A 68.6239,B 3.5749,C 0.0713,E1 3.6397,E2 384.8278} C_DIS
LIN {X 52.1343,Y 132.8498,Z 184,A 70.0189,B 3.5749,C 0.0701,E1 3.6361,E2 383.4392} C_DIS
LIN {X 48.8078,Y 134.1076,Z 184,A 71.4196,B 3.575,C 0.0689,E1 3.6324,E2 382.0422} C_DIS
LIN {X 45.6118,Y 135.2285,Z 184,A 72.7922,B 3.575,C 0.0674,E1 3.6288,E2 380.6682} C_DIS
LIN {X 42.2877,Y 136.3046,Z 184,A 74.3232,B 3.575,C 0.0649,E1 3.6247,E2 379.121} C_DIS
LIN {X 38.0606,Y 137.5443,Z 184,A 75.9233,B 3.575,C 0.0649,E1 3.6204,E2 377.543} C_DIS
LIN {X 34.6606,Y 138.4405,Z 184,A 77.3162,B 3.575,C 0.064,E1 3.6167,E2 376.1529} C_DIS
LIN {X 31.2579,Y 139.2485,Z 184,A 78.7041,B 3.5751,C 0.0631,E1 3.6129,E2 374.7674} C_DIS
LIN {X 27.8368,Y 139.973,Z 184,A 80.0927,B 3.5751,C 0.0623,E1 3.6091,E2 373.3813} C_DIS
LIN {X 24.3986,Y 140.6137,Z 184,A 81.6258,B 3.5751,C 0.0603,E1 3.6049,E2 371.8321} C_DIS
LIN {X 20.9319,Y 141.1714,Z 184,A 82.9055,B 3.5751,C 0.0607,E1 3.6014,E2 370.5695} C_DIS
LIN {X 17.4623,Y 141.6416,Z 184,A 84.2995,B 3.5751,C 0.0602,E1 3.5975,E2 369.1775} C_DIS
LIN {X 13.9835,Y 142.0266,Z 184,A 85.6932,B 3.5751,C 0.0597,E1 3.5936,E2 367.7858} C_DIS
LIN {X 10.4974,Y 142.3264,Z 184,A 87.0856,B 3.5751,C 0.0594,E1 3.5898,E2 366.3954} C_DIS
LIN {X 6.9901,Y 142.5418,Z 184,A 88.4829,B 3.5751,C 0.0591,E1 3.5859,E2 365.0004} C_DIS
LIN {X 3.4941,Y 142.671,Z 184,A 89.8735,B 3.5751,C 0.059,E1 3.582,E2 363.6122} C_DIS
LIN {X -0.0038,Y 142.7152,Z 184,A 91.3168,B 3.5751,C 0.0585,E1 3.5779,E2 362.1645} C_DIS
LIN {X -3.5039,Y 142.6707,Z 184,A 92.8517,B 3.5752,C 0.0574,E1 3.5736,E2 360.6136} C_DIS
LIN {X -7.9254,Y 142.4948,Z 184,A 94.4833,B 3.5752,C 0.0586,E1 3.5691,E2 359.0014} C_DIS
LIN {X -11.4203,Y 142.2565,Z 184,A 95.8733,B 3.5752,C 0.0589,E1 3.5652,E2 357.6142} C_DIS
LIN {X -14.8196,Y 141.9421,Z 184,A 97.2677,B 3.5752,C 0.0589,E1 3.5614,E2 356.2174} C_DIS
LIN {X -18.2959,Y 141.5354,Z 184,A 98.7153,B 3.5752,C 0.059,E1 3.5573,E2 354.765} C_DIS
LIN {X -21.7866,Y 141.04,Z 184,A 100.0913,B 3.5752,C 0.0598,E1 3.5535,E2 353.3948} C_DIS
LIN {X -25.237,Y 140.4636,Z 184,A 101.5136,B 3.5752,C 0.0602,E1 3.5496,E2 351.971} C_DIS
LIN {X -28.7546,Y 139.7862,Z 184,A 103.0356,B 3.5752,C 0.0602,E1 3.5454,E2 350.439} C_DIS
LIN {X -32.9779,Y 138.851,Z 184,A 104.703,B 3.5752,C 0.0616,E1 3.5409,E2 348.7815} C_DIS
LIN {X -36.3619,Y 138.0032,Z 184,A 106.2233,B 3.5752,C 0.0616,E1 3.5367,E2 347.2466} C_DIS
LIN {X -40.5496,Y 136.8314,Z 184,A 107.8825,B 3.5752,C 0.0635,E1 3.5323,E2 345.5996} C_DIS
LIN {X -43.9768,Y 135.7691,Z 184,A 109.4671,B 3.5752,C 0.0635,E1 3.5281,E2 343.9974} C_DIS
LIN {X -48.1052,Y 134.3609,Z 184,A 111.1047,B 3.5751,C 0.0658,E1 3.5238,E2 342.3755} C_DIS
LIN {X -51.3813,Y 133.1426,Z 184,A 112.5254,B 3.5751,C 0.067,E1 3.5201,E2 340.9534} C_DIS
LIN {X -54.6248,Y 131.8452,Z 184,A 114.0341,B 3.5751,C 0.0676,E1 3.5161,E2 339.4319} C_DIS
LIN {X -58.6316,Y 130.1128,Z 184,A 115.7706,B 3.575,C 0.0696,E1 3.5117,E2 337.6986} C_DIS
LIN {X -62.5855,Y 128.2586,Z 184,A 117.5114,B 3.575,C 0.0717,E1 3.5073,E2 335.9607} C_DIS
LIN {X -65.7297,Y 126.6764,Z 184,A 119.0148,B 3.575,C 0.0728,E1 3.5035,E2 334.4466} C_DIS
LIN {X -69.5815,Y 124.6034,Z 184,A 120.8366,B 3.5749,C 0.0746,E1 3.4991,E2 332.6176} C_DIS
LIN {X -73.3777,Y 122.4062,Z 184,A 122.6252,B 3.5749,C 0.0768,E1 3.4948,E2 330.8267} C_DIS
LIN {X -77.0901,Y 120.1023,Z 184,A 124.3888,B 3.5748,C 0.0793,E1 3.4906,E2 329.0631} C_DIS
LIN {X -80.7393,Y 117.68,Z 184,A 126.1952,B 3.5748,C 0.0817,E1 3.4864,E2 327.2519} C_DIS
LIN {X -84.3157,Y 115.1448,Z 184,A 128.0084,B 3.5747,C 0.0841,E1 3.4823,E2 325.4331} C_DIS
LIN {X -87.804,Y 112.5081,Z 184,A 129.8119,B 3.5747,C 0.0867,E1 3.4783,E2 323.6248} C_DIS
LIN {X -91.2094,Y 109.7648,Z 184,A 131.6015,B 3.5745,C 0.0896,E1 3.4744,E2 321.832} C_DIS
LIN {X -94.5424,Y 106.9072,Z 184,A 133.3955,B 3.5745,C 0.0926,E1 3.4706,E2 320.0353} C_DIS
LIN {X -97.7736,Y 103.9605,Z 184,A 135.2196,B 3.5744,C 0.0954,E1 3.4668,E2 318.2038} C_DIS
LIN {X -100.9134,Y 100.9164,Z 184,A 137.0307,B 3.5744,C 0.0985,E1 3.4632,E2 316.3869} C_DIS
LIN {X -103.963,Y 97.771,Z 184,A 138.8305,B 3.5742,C 0.1018,E1 3.4598,E2 314.5831} C_DIS
LIN {X -106.9173,Y 94.5309,Z 184,A 140.6307,B 3.5742,C 0.1052,E1 3.4564,E2 312.7792} C_DIS
LIN {X -109.7617,Y 91.2132,Z 184,A 142.4943,B 3.574,C 0.1083,E1 3.453,E2 310.9028} C_DIS
LIN {X -112.51,Y 87.8015,Z 184,A 144.3185,B 3.574,C 0.1118,E1 3.4498,E2 309.0714} C_DIS
LIN {X -115.3936,Y 83.9751,Z 184,A 146.2645,B 3.5738,C 0.1159,E1 3.4466,E2 307.1241} C_DIS
LIN {X -117.9206,Y 80.3888,Z 184,A 148.096,B 3.5737,C 0.1196,E1 3.4437,E2 305.2849} C_DIS
LIN {X -120.3285,Y 76.7368,Z 184,A 149.8951,B 3.5735,C 0.1235,E1 3.4409,E2 303.4815} C_DIS
LIN {X -122.6228,Y 73.0142,Z 184,A 151.6979,B 3.5734,C 0.1274,E1 3.4383,E2 301.674} C_DIS
LIN {X -124.8022,Y 69.2231,Z 184,A 153.5267,B 3.5733,C 0.1313,E1 3.4358,E2 299.837} C_DIS
LIN {X -126.87,Y 65.3552,Z 184,A 155.3917,B 3.5731,C 0.1351,E1 3.4334,E2 297.9598} C_DIS
LIN {X -128.6402,Y 61.795,Z 184,A 156.9263,B 3.5729,C 0.1395,E1 3.4315,E2 296.4344} C_DIS
LIN {X -130.1165,Y 58.6233,Z 184,A 158.3707,B 3.5729,C 0.1429,E1 3.4298,E2 294.986} C_DIS
LIN {X -131.4967,Y 55.4593,Z 184,A 159.8233,B 3.5727,C 0.1461,E1 3.4282,E2 293.5257} C_DIS
LIN {X -132.849,Y 52.1364,Z 184,A 161.2942,B 3.5725,C 0.1497,E1 3.4267,E2 292.0519} C_DIS
LIN {X -134.0583,Y 48.9447,Z 184,A 162.7452,B 3.5725,C 0.1529,E1 3.4253,E2 290.5915} C_DIS
LIN {X -135.2185,Y 45.642,Z 184,A 164.2076,B 3.5723,C 0.1564,E1 3.4239,E2 289.1227} C_DIS
LIN {X -136.2986,Y 42.3071,Z 184,A 165.8049,B 3.5721,C 0.1591,E1 3.4226,E2 287.5014} C_DIS
LIN {X -137.5439,Y 38.0621,Z 184,A 167.5157,B 3.5719,C 0.1643,E1 3.4213,E2 285.8006} C_DIS
LIN {X -138.4362,Y 34.6775,Z 184,A 168.9766,B 3.5717,C 0.1679,E1 3.4202,E2 284.3335} C_DIS
LIN {X -139.2561,Y 31.2247,Z 184,A 170.5814,B 3.5716,C 0.1709,E1 3.4192,E2 282.7059} C_DIS
LIN {X -140.1332,Y 27.0124,Z 184,A 172.2801,B 3.5713,C 0.1758,E1 3.4183,E2 281.0122} C_DIS
LIN {X -140.9054,Y 22.6555,Z 184,A 174.1241,B 3.5711,C 0.1804,E1 3.4174,E2 279.1608} C_DIS
LIN {X -141.418,Y 19.1918,Z 184,A 175.5873,B 3.5709,C 0.184,E1 3.4169,E2 277.691} C_DIS
LIN {X -141.8452,Y 15.7194,Z 184,A 177.0472,B 3.5707,C 0.1877,E1 3.4164,E2 276.2246} C_DIS
LIN {X -142.1872,Y 12.2403,Z 184,A 178.5043,B 3.5706,C 0.1914,E1 3.416,E2 274.7615} C_DIS
LIN {X -142.4441,Y 8.7553,Z 184,A 179.963,B 3.5704,C 0.195,E1 3.4157,E2 273.2963} C_DIS
LIN {X -142.6172,Y 5.2371,Z 184,A -178.5778,B 3.5701,C 0.1988,E1 3.4156,E2 271.8321} C_DIS
LIN {X -142.7038,Y 1.7427,Z 184,A -177.0154,B 3.57,C 0.2019,E1 3.4155,E2 270.2495} C_DIS
LIN {X -142.7036,Y -1.755,Z 184,A -175.6203,B 3.5697,C 0.2059,E1 3.4155,E2 268.8566} C_DIS
LIN {X -142.5808,Y -6.17,Z 184,A -173.8112,B 3.5695,C 0.2108,E1 3.4157,E2 267.0439} C_DIS
LIN {X -142.3867,Y -9.6704,Z 184,A -172.3071,B 3.5693,C 0.2142,E1 3.4159,E2 265.5278} C_DIS
LIN {X -142.113,Y -13.083,Z 184,A -170.8813,B 3.569,C 0.2178,E1 3.4163,E2 264.0959} C_DIS
LIN {X -141.7489,Y -16.5625,Z 184,A -169.4242,B 3.5688,C 0.2215,E1 3.4167,E2 262.6326} C_DIS
LIN {X -141.2882,Y -20.1149,Z 184,A -167.949,B 3.5686,C 0.2253,E1 3.4173,E2 261.1534} C_DIS
LIN {X -140.6161,Y -24.3852,Z 184,A -166.1162,B 3.5683,C 0.2296,E1 3.4181,E2 259.3086} C_DIS
LIN {X -139.9766,Y -27.8188,Z 184,A -164.6517,B 3.5681,C 0.2331,E1 3.4189,E2 257.8365} C_DIS
LIN {X -139.2466,Y -31.2662,Z 184,A -163.0919,B 3.5679,C 0.2362,E1 3.4199,E2 256.2579} C_DIS
LIN {X -138.2097,Y -35.5698,Z 184,A -161.3547,B 3.5675,C 0.2413,E1 3.421,E2 254.5271} C_DIS
LIN {X -137.3192,Y -38.8655,Z 184,A -159.921,B 3.5673,C 0.2447,E1 3.4221,E2 253.0856} C_DIS
LIN {X -136.299,Y -42.3058,Z 184,A -158.4042,B 3.5671,C 0.2481,E1 3.4233,E2 251.5593} C_DIS
LIN {X -134.9451,Y -46.4413,Z 184,A -156.6066,B 3.5668,C 0.2525,E1 3.4249,E2 249.7557} C_DIS
LIN {X -133.7671,Y -49.7327,Z 184,A -155.1498,B 3.5665,C 0.2559,E1 3.4263,E2 248.2924} C_DIS
LIN {X -132.5092,Y -52.9937,Z 184,A -153.6055,B 3.5663,C 0.2587,E1 3.4279,E2 246.7296} C_DIS
LIN {X -130.8064,Y -57.068,Z 184,A -151.8199,B 3.566,C 0.2632,E1 3.4299,E2 244.9431} C_DIS
LIN {X -129.0113,Y -61.0183,Z 184,A -150.0492,B 3.5657,C 0.2674,E1 3.432,E2 243.1692} C_DIS
LIN {X -127.2877,Y -64.5347,Z 184,A -148.4052,B 3.5654,C 0.271,E1 3.434,E2 241.5161} C_DIS
LIN {X -125.4438,Y -68.0543,Z 184,A -146.6689,B 3.5652,C 0.274,E1 3.4363,E2 239.7612} C_DIS
LIN {X -123.3004,Y -71.8652,Z 184,A -144.8459,B 3.5649,C 0.2779,E1 3.4389,E2 237.9296} C_DIS
LIN {X -121.0409,Y -75.6081,Z 184,A -143.0455,B 3.5646,C 0.2817,E1 3.4415,E2 236.1237} C_DIS
LIN {X -118.662,Y -79.2891,Z 184,A -141.2402,B 3.5643,C 0.2855,E1 3.4443,E2 234.3127} C_DIS
LIN {X -116.0597,Y -83.0516,Z 184,A -139.3655,B 3.564,C 0.2894,E1 3.4473,E2 232.4333} C_DIS
LIN {X -113.5695,Y -86.4263,Z 184,A -137.5802,B 3.5637,C 0.2925,E1 3.4503,E2 230.6345} C_DIS
LIN {X -110.8707,Y -89.8622,Z 184,A -135.7846,B 3.5634,C 0.296,E1 3.4535,E2 228.8337} C_DIS
LIN {X -108.0601,Y -93.2226,Z 184,A -133.9836,B 3.5631,C 0.2994,E1 3.4568,E2 227.0273} C_DIS
LIN {X -105.1522,Y -96.4907,Z 184,A -132.4063,B 3.5627,C 0.304,E1 3.4597,E2 225.4749} C_DIS
LIN {X -103.0428,Y -98.7402,Z 184,A -130.906,B 3.5627,C 0.3048,E1 3.4626,E2 223.9388} C_DIS
LIN {X -99.9565,Y -101.8632,Z 184,A -129.0895,B 3.5624,C 0.3078,E1 3.4662,E2 222.1151} C_DIS
LIN {X -96.7481,Y -104.9156,Z 184,A -127.2641,B 3.5622,C 0.3108,E1 3.47,E2 220.2834} C_DIS
LIN {X -93.5684,Y -107.7613,Z 184,A -125.4836,B 3.5619,C 0.3134,E1 3.4737,E2 218.4938} C_DIS
LIN {X -90.1799,Y -110.6121,Z 184,A -123.691,B 3.5617,C 0.3163,E1 3.4776,E2 216.6993} C_DIS
LIN {X -86.7371,Y -113.3318,Z 184,A -121.8813,B 3.5614,C 0.3188,E1 3.4816,E2 214.883} C_DIS
LIN {X -83.2596,Y -115.9109,Z 184,A -120.0821,B 3.5612,C 0.3211,E1 3.4857,E2 213.0755} C_DIS
LIN {X -79.6331,Y -118.4322,Z 184,A -118.2718,B 3.561,C 0.3235,E1 3.4898,E2 211.26} C_DIS
LIN {X -76.0037,Y -120.7928,Z 184,A -116.5085,B 3.5608,C 0.3258,E1 3.494,E2 209.4932} C_DIS
LIN {X -72.222,Y -123.091,Z 184,A -114.6896,B 3.5606,C 0.3278,E1 3.4984,E2 207.6683} C_DIS
LIN {X -68.4414,Y -125.2326,Z 184,A -112.9658,B 3.5604,C 0.3301,E1 3.5026,E2 205.9473} C_DIS
LIN {X -65.3496,Y -126.8729,Z 184,A -111.4579,B 3.5604,C 0.331,E1 3.5064,E2 204.4249} C_DIS
LIN {X -61.8053,Y -128.6353,Z 184,A -109.961,B 3.5601,C 0.3335,E1 3.5101,E2 202.9407} C_DIS
LIN {X -58.6355,Y -130.1111,Z 184,A -108.5197,B 3.56,C 0.3347,E1 3.5138,E2 201.4939} C_DIS
LIN {X -55.4594,Y -131.4966,Z 184,A -107.1246,B 3.5599,C 0.336,E1 3.5174,E2 200.098} C_DIS
LIN {X -51.7113,Y -133.0143,Z 184,A -105.4143,B 3.5598,C 0.3368,E1 3.5218,E2 198.3753} C_DIS
LIN {X -48.0336,Y -134.3867,Z 184,A -103.883,B 3.5596,C 0.3384,E1 3.5258,E2 196.8499} C_DIS
LIN {X -44.7377,Y -135.5196,Z 184,A -102.4698,B 3.5596,C 0.3394,E1 3.5296,E2 195.4345} C_DIS
LIN {X -41.2503,Y -136.6221,Z 184,A -100.8457,B 3.5596,C 0.3392,E1 3.534,E2 193.7884} C_DIS
LIN {X -37.1687,Y -137.7881,Z 184,A -99.2874,B 3.5594,C 0.3414,E1 3.5381,E2 192.25} C_DIS
LIN {X -33.8635,Y -138.6375,Z 184,A -97.8823,B 3.5594,C 0.3418,E1 3.5419,E2 190.8396} C_DIS
LIN {X -30.0688,Y -139.5091,Z 184,A -96.2494,B 3.5593,C 0.342,E1 3.5464,E2 189.1964} C_DIS
LIN {X -26.124,Y -140.303,Z 184,A -94.697,B 3.5592,C 0.3431,E1 3.5507,E2 187.6524} C_DIS
LIN {X -22.6652,Y -140.9039,Z 184,A -93.2613,B 3.5592,C 0.3434,E1 3.5546,E2 186.2124} C_DIS
LIN {X -19.2015,Y -141.4167,Z 184,A -91.8496,B 3.5592,C 0.3436,E1 3.5585,E2 184.7994} C_DIS
LIN {X -15.7275,Y -141.8444,Z 184,A -90.4435,B 3.5592,C 0.3439,E1 3.5625,E2 183.3927} C_DIS
LIN {X -12.2448,Y -142.1868,Z 184,A -89.0414,B 3.5591,C 0.3441,E1 3.5664,E2 181.9903} C_DIS
LIN {X -8.7416,Y -142.445,Z 184,A -87.6376,B 3.5591,C 0.3441,E1 3.5703,E2 180.5868} C_DIS
LIN {X -4.9895,Y -142.6269,Z 184,A -86.0085,B 3.5591,C 0.3431,E1 3.5749,E2 178.9402} C_DIS
LIN {X 0.0014,Y -142.7152,Z 184,A -84.1038,B 3.5591,C 0.3437,E1 3.5802,E2 177.0484} C_DIS
LIN {X 0.0014,Y -142.7152,Z 184,A -84.1038,B 3.5591,C 0.3437,E1 3.5802,E2 177.0484} C_DIS
Enddeposition()
LIN {X 0.9683,Y -133.7631,Z 185,A -83.8534,B 3.0783,C 0.3105,E1 3.0989,E2 176.6446} C_DIS
Startdeposition()
$VEL.CP = VEL_PRINT
LIN {X -1.6595,Y -133.7584,Z 185,A -85.249,B 3.0781,C 0.3126,E1 3.0949,E2 178.0757} C_DIS
LIN {X -4.8428,Y -133.6802,Z 185,A -86.6298,B 3.0781,C 0.3129,E1 3.0911,E2 179.4593} C_DIS
LIN {X -8.2074,Y -133.5153,Z 185,A -87.9839,B 3.0781,C 0.3123,E1 3.0873,E2 180.8026} C_DIS
LIN {X -11.2591,Y -133.2927,Z 185,A -89.4056,B 3.0781,C 0.313,E1 3.0833,E2 182.2391} C_DIS
LIN {X -14.7399,Y -132.9534,Z 185,A -90.8666,B 3.0781,C 0.3125,E1 3.0793,E2 183.696} C_DIS
LIN {X -18.0088,Y -132.551,Z 185,A -92.2752,B 3.0781,C 0.3123,E1 3.0754,E2 185.1048} C_DIS
LIN {X -21.1632,Y -132.0844,Z 185,A -93.6814,B 3.0781,C 0.3122,E1 3.0715,E2 186.5168} C_DIS
LIN {X -24.4862,Y -131.5085,Z 185,A -95.1235,B 3.0781,C 0.3117,E1 3.0675,E2 187.9591} C_DIS
LIN {X -27.7032,Y -130.8681,Z 185,A -96.5355,B 3.0782,C 0.3112,E1 3.0636,E2 189.3724} C_DIS
LIN {X -30.9119,Y -130.1472,Z 185,A -97.9527,B 3.0782,C 0.3105,E1 3.0598,E2 190.7912} C_DIS
LIN {X -33.7775,Y -129.4342,Z 185,A -99.3013,B 3.0782,C 0.3104,E1 3.0561,E2 192.151} C_DIS
LIN {X -37.1677,Y -128.5005,Z 185,A -100.7737,B 3.0784,C 0.3093,E1 3.0521,E2 193.6194} C_DIS
LIN {X -40.3962,Y -127.522,Z 185,A -102.1825,B 3.0785,C 0.3081,E1 3.0484,E2 195.0239} C_DIS
LIN {X -44.1833,Y -126.26,Z 185,A -103.974,B 3.0785,C 0.3073,E1 3.0436,E2 196.8263} C_DIS
LIN {X -48.0602,Y -124.8359,Z 185,A -105.7308,B 3.0788,C 0.3057,E1 3.039,E2 198.5819} C_DIS
LIN {X -50.7321,Y -123.7758,Z 185,A -107.0948,B 3.0788,C 0.3054,E1 3.0354,E2 199.9632} C_DIS
LIN {X -54.2098,Y -122.2909,Z 185,A -108.595,B 3.079,C 0.3031,E1 3.0316,E2 201.4483} C_DIS
LIN {X -57.1081,Y -120.9653,Z 185,A -110.0119,B 3.0791,C 0.302,E1 3.028,E2 202.8721} C_DIS
LIN {X -60.0549,Y -119.5302,Z 185,A -111.4741,B 3.0792,C 0.3008,E1 3.0243,E2 204.342} C_DIS
LIN {X -63.06,Y -117.973,Z 185,A -112.8433,B 3.0794,C 0.2987,E1 3.021,E2 205.701} C_DIS
LIN {X -65.9478,Y -116.3837,Z 185,A -114.3444,B 3.0796,C 0.2974,E1 3.0173,E2 207.2137} C_DIS
LIN {X -68.6916,Y -114.7851,Z 185,A -115.7602,B 3.0797,C 0.2959,E1 3.0138,E2 208.6367} C_DIS
LIN {X -71.5684,Y -113.0138,Z 185,A -117.2317,B 3.0799,C 0.2941,E1 3.0103,E2 210.1114} C_DIS
LIN {X -74.2382,Y -111.278,Z 185,A -118.6539,B 3.08,C 0.2925,E1 3.007,E2 211.541} C_DIS
LIN {X -77.0209,Y -109.3705,Z 185,A -120.114,B 3.0802,C 0.2904,E1 3.0036,E2 213.0031} C_DIS
LIN {X -79.6029,Y -107.5063,Z 185,A -121.5363,B 3.0804,C 0.2886,E1 3.0004,E2 214.4328} C_DIS
LIN {X -82.2679,Y -105.4811,Z 185,A -122.9965,B 3.0806,C 0.2864,E1 2.9972,E2 215.8964} C_DIS
LIN {X -84.8297,Y -103.4316,Z 185,A -124.4453,B 3.0808,C 0.2843,E1 2.994,E2 217.3506} C_DIS
LIN {X -87.9598,Y -100.7828,Z 185,A -126.2513,B 3.0811,C 0.2815,E1 2.9902,E2 219.1629} C_DIS
LIN {X -91.0077,Y -98.0395,Z 185,A -128.0615,B 3.0813,C 0.2786,E1 2.9864,E2 220.9797} C_DIS
LIN {X -93.9775,Y -95.1973,Z 185,A -129.8815,B 3.0816,C 0.2756,E1 2.9827,E2 222.807} C_DIS
LIN {X -96.3465,Y -92.7986,Z 185,A -131.5206,B 3.0818,C 0.2738,E1 2.9795,E2 224.4706} C_DIS
LIN {X -99.6361,Y -89.2567,Z 185,A -133.5111,B 3.0822,C 0.2693,E1 2.9758,E2 226.4506} C_DIS
LIN {X -101.2915,Y -87.3737,Z 185,A -134.7605,B 3.0822,C 0.2679,E1 2.9735,E2 227.722} C_DIS
LIN {X -103.9229,Y -84.2274,Z 185,A -136.4252,B 3.0826,C 0.2638,E1 2.9705,E2 229.3747} C_DIS
LIN {X -105.957,Y -81.6539,Z 185,A -138.0437,B 3.0828,C 0.2617,E1 2.9677,E2 231.0198} C_DIS
LIN {X -108.4086,Y -78.3691,Z 185,A -139.6969,B 3.0832,C 0.2574,E1 2.965,E2 232.6596} C_DIS
LIN {X -110.2495,Y -75.7573,Z 185,A -141.134,B 3.0834,C 0.2546,E1 2.9627,E2 234.105} C_DIS
LIN {X -112.1306,Y -72.9442,Z 185,A -142.6127,B 3.0837,C 0.2514,E1 2.9604,E2 235.5869} C_DIS
LIN {X -113.8356,Y -70.2545,Z 185,A -144.0807,B 3.0839,C 0.2487,E1 2.9582,E2 237.0676} C_DIS
LIN {X -115.1959,Y -68.0008,Z 185,A -145.3762,B 3.084,C 0.2467,E1 2.9563,E2 238.3837} C_DIS
LIN {X -117.1476,Y -64.5803,Z 185,A -146.9922,B 3.0844,C 0.2423,E1 2.9541,E2 239.9903} C_DIS
LIN {X -118.6916,Y -61.6942,Z 185,A -148.4571,B 3.0846,C 0.2392,E1 2.9522,E2 241.4625} C_DIS
LIN {X -120.2131,Y -58.6744,Z 185,A -149.9671,B 3.0849,C 0.2358,E1 2.9503,E2 242.9797} C_DIS
LIN {X -121.6159,Y -55.7079,Z 185,A -151.4328,B 3.0851,C 0.2325,E1 2.9486,E2 244.4523} C_DIS
LIN {X -122.9105,Y -52.7891,Z 185,A -152.8694,B 3.0854,C 0.2293,E1 2.947,E2 245.897} C_DIS
LIN {X -124.2037,Y -49.6706,Z 185,A -154.3552,B 3.0856,C 0.2257,E1 2.9454,E2 247.3871} C_DIS
LIN {X -125.3864,Y -46.6043,Z 185,A -155.839,B 3.0859,C 0.2224,E1 2.9439,E2 248.8797} C_DIS
LIN {X -126.4605,Y -43.605,Z 185,A -157.2849,B 3.0861,C 0.2191,E1 2.9426,E2 250.3351} C_DIS
LIN {X -127.5301,Y -40.3708,Z 185,A -158.7776,B 3.0864,C 0.2153,E1 2.9413,E2 251.8313} C_DIS
LIN {X -128.3003,Y -37.8515,Z 185,A -160.0342,B 3.0866,C 0.2128,E1 2.9403,E2 253.1033} C_DIS
LIN {X -129.3504,Y -34.0916,Z 185,A -161.7099,B 3.0869,C 0.2083,E1 2.939,E2 254.7785} C_DIS
LIN {X -130.1261,Y -30.9992,Z 185,A -163.1494,B 3.0871,C 0.2048,E1 2.9381,E2 256.2264} C_DIS
LIN {X -130.8473,Y -27.7996,Z 185,A -164.6195,B 3.0873,C 0.2012,E1 2.9372,E2 257.7039} C_DIS
LIN {X -131.4903,Y -24.5815,Z 185,A -166.0897,B 3.0876,C 0.1976,E1 2.9364,E2 259.1813} C_DIS
LIN {X -132.0558,Y -21.3401,Z 185,A -167.5894,B 3.0878,C 0.194,E1 2.9357,E2 260.6913} C_DIS
LIN {X -132.5515,Y -18.0045,Z 185,A -169.0707,B 3.088,C 0.1901,E1 2.9351,E2 262.1763} C_DIS
LIN {X -132.9427,Y -14.8395,Z 185,A -170.5336,B 3.0883,C 0.1866,E1 2.9346,E2 263.6504} C_DIS
LIN {X -133.266,Y -11.5742,Z 185,A -171.9482,B 3.0885,C 0.1827,E1 2.9343,E2 265.0652} C_DIS
LIN {X -133.51,Y -8.2944,Z 185,A -173.342,B 3.0887,C 0.1787,E1 2.934,E2 266.4563} C_DIS
LIN {X -133.6771,Y -4.9229,Z 185,A -174.9777,B 3.0889,C 0.1753,E1 2.9338,E2 268.1144} C_DIS
LIN {X -133.7586,Y -1.6435,Z 185,A -176.4057,B 3.0891,C 0.1714,E1 2.9337,E2 269.5443} C_DIS
LIN {X -133.7631,Y 1.2189,Z 185,A -177.8212,B 3.0893,C 0.1686,E1 2.9337,E2 270.9821} C_DIS
LIN {X -133.6806,Y 4.8339,Z 185,A -179.387,B 3.0895,C 0.1643,E1 2.9338,E2 272.549} C_DIS
LIN {X -133.5466,Y 7.6995,Z 185,A 179.2069,B 3.0897,C 0.1615,E1 2.9341,E2 273.9759} C_DIS
LIN {X -133.2745,Y 11.4745,Z 185,A 177.6405,B 3.0899,C 0.1567,E1 2.9344,E2 275.5345} C_DIS
LIN {X -132.9533,Y 14.7409,Z 185,A 176.17,B 3.0901,C 0.153,E1 2.9348,E2 277.0119} C_DIS
LIN {X -132.5526,Y 17.996,Z 185,A 174.7023,B 3.0903,C 0.1493,E1 2.9354,E2 278.4863} C_DIS
LIN {X -132.085,Y 21.1593,Z 185,A 173.2316,B 3.0904,C 0.1459,E1 2.936,E2 279.9683} C_DIS
LIN {X -131.5089,Y 24.4842,Z 185,A 171.7886,B 3.0906,C 0.1418,E1 2.9367,E2 281.41} C_DIS
LIN {X -130.8478,Y 27.7975,Z 185,A 170.2241,B 3.0908,C 0.1382,E1 2.9376,E2 282.9876} C_DIS
LIN {X -130.1409,Y 30.9381,Z 185,A 168.774,B 3.0909,C 0.1347,E1 2.9385,E2 284.4453} C_DIS
LIN {X -129.4174,Y 33.8405,Z 185,A 167.3786,B 3.0911,C 0.1316,E1 2.9395,E2 285.8535} C_DIS
LIN {X -128.4982,Y 37.1753,Z 185,A 165.8517,B 3.0912,C 0.1278,E1 2.9406,E2 287.3847} C_DIS
LIN {X -127.5209,Y 40.3996,Z 185,A 164.3962,B 3.0914,C 0.1239,E1 2.9418,E2 288.8407} C_DIS
LIN {X -126.5237,Y 43.4226,Z 185,A 162.9126,B 3.0915,C 0.1207,E1 2.9432,E2 290.3377} C_DIS
LIN {X -125.4177,Y 46.5208,Z 185,A 161.4696,B 3.0917,C 0.1171,E1 2.9445,E2 291.7838} C_DIS
LIN {X -124.2396,Y 49.5815,Z 185,A 160.0023,B 3.0917,C 0.1137,E1 2.946,E2 293.2575} C_DIS
LIN {X -122.987,Y 52.6121,Z 185,A 158.5057,B 3.0919,C 0.1104,E1 2.9477,E2 294.7641} C_DIS
LIN {X -121.661,Y 55.6104,Z 185,A 157.0715,B 3.092,C 0.1069,E1 2.9493,E2 296.2007} C_DIS
LIN {X -120.2562,Y 58.5872,Z 185,A 155.6582,B 3.0922,C 0.1033,E1 2.951,E2 297.6134} C_DIS
LIN {X -118.7354,Y 61.6109,Z 185,A 154.106,B 3.0922,C 0.1001,E1 2.953,E2 299.1767} C_DIS
LIN {X -117.1885,Y 64.5064,Z 185,A 152.6211,B 3.0924,C 0.097,E1 2.955,E2 300.6699} C_DIS
LIN {X -115.6198,Y 67.2774,Z 185,A 151.1901,B 3.0924,C 0.0939,E1 2.957,E2 302.1079} C_DIS
LIN {X -113.9354,Y 70.0919,Z 185,A 149.7135,B 3.0925,C 0.0908,E1 2.9591,E2 303.5919} C_DIS
LIN {X -112.1185,Y 72.9629,Z 185,A 148.2324,B 3.0926,C 0.0875,E1 2.9614,E2 305.0749} C_DIS
LIN {X -110.2973,Y 75.6877,Z 185,A 146.7586,B 3.0927,C 0.0846,E1 2.9637,E2 306.556} C_DIS
LIN {X -108.5069,Y 78.2335,Z 185,A 145.3595,B 3.0927,C 0.0818,E1 2.966,E2 307.9619} C_DIS
LIN {X -106.4597,Y 80.9973,Z 185,A 143.8574,B 3.0929,C 0.0787,E1 2.9685,E2 309.4663} C_DIS
LIN {X -104.2576,Y 83.8123,Z 185,A 142.1269,B 3.0929,C 0.0761,E1 2.9715,E2 311.2192} C_DIS
LIN {X -101.2497,Y 87.4222,Z 185,A 140.0104,B 3.093,C 0.0723,E1 2.9754,E2 313.3464} C_DIS
LIN {X -98.0409,Y 91.0062,Z 185,A 137.8874,B 3.0931,C 0.0684,E1 2.9794,E2 315.4752} C_DIS
LIN {X -95.2158,Y 93.9586,Z 185,A 136.0786,B 3.0931,C 0.0652,E1 2.9829,E2 317.2896} C_DIS
LIN {X -92.2066,Y 96.9131,Z 185,A 134.2013,B 3.0933,C 0.0621,E1 2.9867,E2 319.1738} C_DIS
LIN {X -88.6507,Y 100.1757,Z 185,A 132.1755,B 3.0933,C 0.0581,E1 2.9909,E2 321.1932} C_DIS
LIN {X -85.4137,Y 102.9496,Z 185,A 130.1998,B 3.0933,C 0.0556,E1 2.9952,E2 323.1851} C_DIS
LIN {X -81.6205,Y 105.9829,Z 185,A 128.0562,B 3.0934,C 0.0524,E1 2.9999,E2 325.3347} C_DIS
LIN {X -78.3566,Y 108.4177,Z 185,A 126.4324,B 3.0934,C 0.0491,E1 3.0035,E2 326.9431} C_DIS
LIN {X -75.7661,Y 110.2434,Z 185,A 125.0183,B 3.0935,C 0.0473,E1 3.0068,E2 328.3629} C_DIS
LIN {X -72.9361,Y 112.1358,Z 185,A 123.5554,B 3.0935,C 0.0452,E1 3.0102,E2 329.8253} C_DIS
LIN {X -70.2458,Y 113.8409,Z 185,A 122.112,B 3.0935,C 0.0436,E1 3.0136,E2 331.2771} C_DIS
LIN {X -67.3559,Y 115.5744,Z 185,A 120.6566,B 3.0935,C 0.0417,E1 3.0171,E2 332.7329} C_DIS
LIN {X -64.5861,Y 117.1444,Z 185,A 119.2593,B 3.0936,C 0.0401,E1 3.0205,E2 334.1332} C_DIS
LIN {X -62.1225,Y 118.4667,Z 185,A 117.9669,B 3.0936,C 0.0391,E1 3.0237,E2 335.4358} C_DIS
LIN {X -58.6703,Y 120.2151,Z 185,A 116.344,B 3.0936,C 0.037,E1 3.0278,E2 337.0536} C_DIS
LIN {X -55.7057,Y 121.6169,Z 185,A 114.9148,B 3.0936,C 0.0356,E1 3.0314,E2 338.4847} C_DIS
LIN {X -52.7452,Y 122.9295,Z 185,A 113.4966,B 3.0936,C 0.0344,E1 3.0351,E2 339.9057} C_DIS
LIN {X -49.6468,Y 124.2132,Z 185,A 112.047,B 3.0937,C 0.0331,E1 3.0388,E2 341.3559} C_DIS
LIN {X -46.5971,Y 125.3891,Z 185,A 110.6264,B 3.0937,C 0.0319,E1 3.0425,E2 342.7781} C_DIS
LIN {X -43.6043,Y 126.4608,Z 185,A 109.2341,B 3.0937,C 0.031,E1 3.0462,E2 344.173} C_DIS
LIN {X -40.4091,Y 127.5179,Z 185,A 107.7999,B 3.0937,C 0.0298,E1 3.05,E2 345.6056} C_DIS
LIN {X -37.3452,Y 128.4485,Z 185,A 106.4574,B 3.0937,C 0.0287,E1 3.0536,E2 346.9439} C_DIS
LIN {X -34.0927,Y 129.3501,Z 185,A 104.9506,B 3.0937,C 0.0282,E1 3.0577,E2 348.457} C_DIS
LIN {X -30.9995,Y 130.1261,Z 185,A 103.6474,B 3.0937,C 0.027,E1 3.0612,E2 349.7521} C_DIS
LIN {X -27.7869,Y 130.8501,Z 185,A 102.1429,B 3.0937,C 0.027,E1 3.0653,E2 351.2668} C_DIS
LIN {X -24.5702,Y 131.4925,Z 185,A 100.7311,B 3.0937,C 0.0264,E1 3.0692,E2 352.6786} C_DIS
LIN {X -21.3389,Y 132.056,Z 185,A 99.2958,B 3.0937,C 0.026,E1 3.0732,E2 354.1167} C_DIS
LIN {X -18.0045,Y 132.5515,Z 185,A 97.9326,B 3.0937,C 0.0252,E1 3.0769,E2 355.4699} C_DIS
LIN {X -14.8237,Y 132.9444,Z 185,A 96.4703,B 3.0937,C 0.0254,E1 3.081,E2 356.9418} C_DIS
LIN {X -11.5614,Y 133.2671,Z 185,A 95.0672,B 3.0937,C 0.0252,E1 3.0849,E2 358.3441} C_DIS
LIN {X -8.7861,Y 133.4797,Z 185,A 93.7572,B 3.0937,C 0.0259,E1 3.0886,E2 359.6673} C_DIS
LIN {X -4.9234,Y 133.6771,Z 185,A 92.287,B 3.0937,C 0.0247,E1 3.0927,E2 361.1151} C_DIS
LIN {X -1.627,Y 133.7589,Z 185,A 90.8398,B 3.0937,C 0.025,E1 3.0967,E2 362.5658} C_DIS
LIN {X 1.6521,Y 133.7585,Z 185,A 89.4206,B 3.0937,C 0.0253,E1 3.1007,E2 363.9861} C_DIS
LIN {X 4.8355,Y 133.6805,Z 185,A 88.0412,B 3.0937,C 0.0257,E1 3.1045,E2 365.3667} C_DIS
LIN {X 8.2034,Y 133.5156,Z 185,A 86.4586,B 3.0937,C 0.027,E1 3.109,E2 366.9648} C_DIS
LIN {X 13.1188,Y 133.1229,Z 185,A 84.5225,B 3.0937,C 0.0266,E1 3.1143,E2 368.8797} C_DIS
LIN {X 16.3801,Y 132.7617,Z 185,A 83.1304,B 3.0937,C 0.0271,E1 3.1182,E2 370.2698} C_DIS
LIN {X 19.5385,Y 132.3341,Z 185,A 81.7767,B 3.0937,C 0.0277,E1 3.1219,E2 371.6217} C_DIS
LIN {X 22.8693,Y 131.7997,Z 185,A 80.3244,B 3.0937,C 0.0286,E1 3.126,E2 373.0744} C_DIS
LIN {X 25.6781,Y 131.2807,Z 185,A 79.0369,B 3.0937,C 0.0299,E1 3.1295,E2 374.369} C_DIS
LIN {X 29.3104,Y 130.5173,Z 185,A 77.677,B 3.0937,C 0.0293,E1 3.1331,E2 375.7016} C_DIS
LIN {X 32.5027,Y 129.7589,Z 185,A 76.1611,B 3.0937,C 0.0312,E1 3.1373,E2 377.23} C_DIS
LIN {X 35.5856,Y 128.9477,Z 185,A 74.8156,B 3.0937,C 0.0322,E1 3.1409,E2 378.5729} C_DIS
LIN {X 38.8279,Y 128.0083,Z 185,A 73.2637,B 3.0937,C 0.0343,E1 3.1451,E2 380.1368} C_DIS
LIN {X 43.2759,Y 126.5746,Z 185,A 71.3519,B 3.0937,C 0.0357,E1 3.1502,E2 382.0377} C_DIS
LIN {X 46.5219,Y 125.4172,Z 185,A 70.0782,B 3.0937,C 0.0357,E1 3.1534,E2 383.2874} C_DIS
LIN {X 49.5871,Y 124.2373,Z 185,A 68.5947,B 3.0937,C 0.0379,E1 3.1573,E2 384.7797} C_DIS
LIN {X 52.6185,Y 122.9843,Z 185,A 67.1903,B 3.0937,C 0.0395,E1 3.161,E2 386.1838} C_DIS
LIN {X 55.6166,Y 121.6582,Z 185,A 65.8436,B 3.0937,C 0.0409,E1 3.1644,E2 387.5236} C_DIS
LIN {X 58.5837,Y 120.2579,Z 185,A 64.4675,B 3.0936,C 0.0425,E1 3.1678,E2 388.8962} C_DIS
LIN {X 61.4979,Y 118.7947,Z 185,A 63.0699,B 3.0936,C 0.0444,E1 3.1713,E2 390.2937} C_DIS
LIN {X 64.5161,Y 117.1831,Z 185,A 61.7806,B 3.0936,C 0.0451,E1 3.1744,E2 391.5622} C_DIS
LIN {X 67.2676,Y 115.6255,Z 185,A 60.3385,B 3.0936,C 0.0478,E1 3.178,E2 393.0146} C_DIS
LIN {X 70.0958,Y 113.933,Z 185,A 58.9514,B 3.0935,C 0.0498,E1 3.1813,E2 394.3987} C_DIS
LIN {X 72.9445,Y 112.1304,Z 185,A 57.5765,B 3.0935,C 0.0516,E1 3.1845,E2 395.7655} C_DIS
LIN {X 75.6729,Y 110.3074,Z 185,A 56.1944,B 3.0935,C 0.0537,E1 3.1877,E2 397.1448} C_DIS
LIN {X 78.3621,Y 108.4136,Z 185,A 54.8513,B 3.0934,C 0.0556,E1 3.1907,E2 398.4801} C_DIS
LIN {X 81.0035,Y 106.455,Z 185,A 53.469,B 3.0934,C 0.0578,E1 3.1938,E2 399.8594} C_DIS
LIN {X 83.5907,Y 104.4358,Z 185,A 51.9391,B 3.0933,C 0.0614,E1 3.1972,E2 401.4041} C_DIS
LIN {X 86.7515,Y 101.8249,Z 185,A 50.3925,B 3.0933,C 0.063,E1 3.2004,E2 402.926} C_DIS
LIN {X 89.2364,Y 99.6543,Z 185,A 48.8775,B 3.0932,C 0.0666,E1 3.2036,E2 404.4532} C_DIS
LIN {X 92.244,Y 96.8773,Z 185,A 47.1862,B 3.0931,C 0.0695,E1 3.2071,E2 406.1373} C_DIS
LIN {X 95.1656,Y 94.0094,Z 185,A 45.6145,B 3.0931,C 0.0715,E1 3.2101,E2 407.6877} C_DIS
LIN {X 97.4819,Y 91.6049,Z 185,A 44.1012,B 3.093,C 0.0752,E1 3.2131,E2 409.2112} C_DIS
LIN {X 100.1804,Y 88.6454,Z 185,A 42.5754,B 3.093,C 0.0773,E1 3.2159,E2 410.7147} C_DIS
LIN {X 102.8506,Y 85.5333,Z 185,A 40.8825,B 3.0928,C 0.0805,E1 3.2189,E2 412.4004} C_DIS
LIN {X 104.945,Y 82.9507,Z 185,A 39.5101,B 3.0928,C 0.0833,E1 3.2213,E2 413.767} C_DIS
LIN {X 107.388,Y 79.7618,Z 185,A 37.8398,B 3.0927,C 0.0868,E1 3.2241,E2 415.4316} C_DIS
LIN {X 109.3199,Y 77.0927,Z 185,A 36.4981,B 3.0926,C 0.0894,E1 3.2263,E2 416.7654} C_DIS
LIN {X 111.176,Y 74.391,Z 185,A 35.1288,B 3.0926,C 0.0924,E1 3.2284,E2 418.1309} C_DIS
LIN {X 112.9658,Y 71.6445,Z 185,A 33.8388,B 3.0924,C 0.0947,E1 3.2303,E2 419.4076} C_DIS
LIN {X 114.7357,Y 68.7747,Z 185,A 32.4124,B 3.0924,C 0.0981,E1 3.2324,E2 420.8324} C_DIS
LIN {X 116.0962,Y 66.4516,Z 185,A 31.209,B 3.0922,C 0.1014,E1 3.2341,E2 422.0422} C_DIS
LIN {X 117.9285,Y 63.1429,Z 185,A 29.7119,B 3.0922,C 0.1043,E1 3.2361,E2 423.5251} C_DIS
LIN {X 119.4414,Y 60.2294,Z 185,A 28.3803,B 3.092,C 0.1072,E1 3.2378,E2 424.8481} C_DIS
LIN {X 120.9273,Y 57.1877,Z 185,A 26.9971,B 3.092,C 0.1103,E1 3.2394,E2 426.2238} C_DIS
LIN {X 122.2925,Y 54.2063,Z 185,A 25.66,B 3.0918,C 0.1133,E1 3.241,E2 427.5533} C_DIS
LIN {X 123.5846,Y 51.1917,Z 185,A 24.3054,B 3.0917,C 0.1165,E1 3.2424,E2 428.9024} C_DIS
LIN {X 124.8095,Y 48.128,Z 185,A 22.9528,B 3.0916,C 0.1196,E1 3.2438,E2 430.2483} C_DIS
LIN {X 125.9457,Y 45.0707,Z 185,A 21.6268,B 3.0915,C 0.1226,E1 3.2451,E2 431.5663} C_DIS
LIN {X 127.015,Y 41.9631,Z 185,A 20.2663,B 3.0913,C 0.126,E1 3.2463,E2 432.9217} C_DIS
LIN {X 127.9793,Y 38.9225,Z 185,A 18.9964,B 3.0913,C 0.1287,E1 3.2473,E2 434.1806} C_DIS
LIN {X 128.922,Y 35.6775,Z 185,A 17.5746,B 3.091,C 0.1324,E1 3.2484,E2 435.6} C_DIS
LIN {X 129.7358,Y 32.5937,Z 185,A 16.2679,B 3.091,C 0.1356,E1 3.2493,E2 436.9001} C_DIS
LIN {X 130.4964,Y 29.4021,Z 185,A 14.9251,B 3.0908,C 0.1389,E1 3.2502,E2 438.236} C_DIS
LIN {X 131.181,Y 26.1811,Z 185,A 13.5782,B 3.0906,C 0.1421,E1 3.2509,E2 439.576} C_DIS
LIN {X 131.7839,Y 22.9573,Z 185,A 12.238,B 3.0905,C 0.1454,E1 3.2516,E2 440.909} C_DIS
LIN {X 132.3213,Y 19.6277,Z 185,A 10.8346,B 3.0903,C 0.149,E1 3.2522,E2 442.3082} C_DIS
LIN {X 132.7508,Y 16.4712,Z 185,A 9.5301,B 3.0901,C 0.1523,E1 3.2526,E2 443.6061} C_DIS
LIN {X 133.1148,Y 13.2034,Z 185,A 8.2505,B 3.0901,C 0.155,E1 3.253,E2 444.8708} C_DIS
LIN {X 133.3987,Y 9.9262,Z 185,A 6.8464,B 3.0898,C 0.1589,E1 3.2533,E2 446.2751} C_DIS
LIN {X 133.6018,Y 6.6547,Z 185,A 5.4991,B 3.0896,C 0.1623,E1 3.2535,E2 447.6163} C_DIS
LIN {X 133.7278,Y 3.2854,Z 185,A 4.1441,B 3.0895,C 0.1655,E1 3.2537,E2 448.9612} C_DIS
LIN {X 133.7704,Y -0.0232,Z 185,A 2.7764,B 3.0893,C 0.169,E1 3.2537,E2 450.3238} C_DIS
LIN {X 133.7302,Y -3.199,Z 185,A 1.458,B 3.0891,C 0.1724,E1 3.2537,E2 451.6379} C_DIS
LIN {X 133.6109,Y -6.4737,Z 185,A 0.1392,B 3.0889,C 0.1756,E1 3.2535,E2 452.947} C_DIS
LIN {X 133.405,Y -9.8397,Z 185,A -1.2461,B 3.0887,C 0.179,E1 3.2532,E2 454.3261} C_DIS
LIN {X 133.181,Y -12.5132,Z 185,A -2.4494,B 3.0885,C 0.1828,E1 3.2529,E2 455.5368} C_DIS
LIN {X 132.7616,Y -16.3804,Z 185,A -3.9299,B 3.0883,C 0.1857,E1 3.2524,E2 456.9955} C_DIS
LIN {X 132.3343,Y -19.5369,Z 185,A -5.2344,B 3.0881,C 0.1889,E1 3.2519,E2 458.2935} C_DIS
LIN {X 131.7997,Y -22.8692,Z 185,A -6.6367,B 3.0879,C 0.1925,E1 3.2513,E2 459.6915} C_DIS
LIN {X 131.1987,Y -26.0939,Z 185,A -7.9779,B 3.0877,C 0.1958,E1 3.2506,E2 461.0258} C_DIS
LIN {X 130.519,Y -29.3032,Z 185,A -9.32,B 3.0875,C 0.1991,E1 3.2498,E2 462.361} C_DIS
LIN {X 129.7841,Y -32.4037,Z 185,A -10.6529,B 3.0873,C 0.2025,E1 3.2489,E2 463.691} C_DIS
LIN {X 128.9474,Y -35.5865,Z 185,A -11.9727,B 3.0871,C 0.2055,E1 3.248,E2 465.0006} C_DIS
LIN {X 128.0083,Y -38.8279,Z 185,A -13.3552,B 3.0868,C 0.2088,E1 3.2469,E2 466.3763} C_DIS
LIN {X 127.047,Y -41.8669,Z 185,A -14.6688,B 3.0866,C 0.212,E1 3.2458,E2 467.6844} C_DIS
LIN {X 126.0127,Y -44.885,Z 185,A -15.9985,B 3.0864,C 0.2153,E1 3.2445,E2 469.0106} C_DIS
LIN {X 124.9433,Y -47.7839,Z 185,A -17.3199,B 3.0861,C 0.2188,E1 3.2432,E2 470.3328} C_DIS
LIN {X 123.6271,Y -51.0899,Z 185,A -18.7022,B 3.086,C 0.2215,E1 3.2418,E2 471.6985} C_DIS
LIN {X 122.2912,Y -54.2093,Z 185,A -20.061,B 3.0857,C 0.2243,E1 3.2403,E2 473.0464} C_DIS
LIN {X 120.9653,Y -57.1081,Z 185,A -21.3962,B 3.0855,C 0.2276,E1 3.2387,E2 474.3789} C_DIS
LIN {X 119.7934,Y -59.5252,Z 185,A -22.6149,B 3.0852,C 0.2312,E1 3.2372,E2 475.6071} C_DIS
LIN {X 117.9653,Y -63.0744,Z 185,A -24.1433,B 3.085,C 0.2338,E1 3.2353,E2 477.114} C_DIS
LIN {X 116.3858,Y -65.944,Z 185,A -25.427,B 3.0849,C 0.2362,E1 3.2335,E2 478.3838} C_DIS
LIN {X 114.7838,Y -68.6938,Z 185,A -26.8077,B 3.0846,C 0.2397,E1 3.2316,E2 479.7677} C_DIS
LIN {X 113.0171,Y -71.5632,Z 185,A -28.1948,B 3.0844,C 0.2427,E1 3.2295,E2 481.149} C_DIS
LIN {X 111.2828,Y -74.231,Z 185,A -29.5206,B 3.0841,C 0.2456,E1 3.2275,E2 482.4711} C_DIS
Enddeposition()
END
